C05492=1189.605,68.219,-48.419,-179.170,5.909,148.807
C05493=1189.600,68.469,-48.436,-179.167,5.909,148.806
C05494=1189.595,68.718,-48.452,-179.164,5.911,148.806
C05495=1189.590,68.967,-48.469,-179.162,5.911,148.805
C05496=1189.585,69.217,-48.486,-179.160,5.912,148.805
C05497=1189.581,69.466,-48.504,-179.157,5.913,148.804
C05498=1189.575,69.715,-48.520,-179.154,5.914,148.804
C05499=1189.570,69.965,-48.538,-179.152,5.915,148.803
C05500=1189.566,70.214,-48.554,-179.149,5.916,148.802
C05501=1189.561,70.464,-48.572,-179.146,5.917,148.802
C05502=1189.555,70.713,-48.588,-179.144,5.918,148.801
C05503=1189.551,70.962,-48.604,-179.142,5.919,148.801
C05504=1189.546,71.211,-48.622,-179.138,5.920,148.800
C05505=1189.542,71.461,-48.639,-179.136,5.921,148.800
C05506=1189.536,71.710,-48.656,-179.134,5.922,148.799
C05507=1189.531,71.960,-48.673,-179.130,5.923,148.798
C05508=1189.526,72.209,-48.690,-179.128,5.924,148.798
C05509=1189.521,72.458,-48.708,-179.126,5.924,148.797
C05510=1189.517,72.708,-48.725,-179.123,5.926,148.797
C05511=1189.511,72.957,-48.742,-179.120,5.927,148.796
C05512=1189.506,73.206,-48.758,-179.118,5.927,148.796
C05513=1189.501,73.456,-48.776,-179.115,5.928,148.795
C05514=1189.497,73.705,-48.793,-179.112,5.929,148.794
C05515=1189.492,73.955,-48.810,-179.110,5.930,148.794
C05516=1189.487,74.204,-48.827,-179.107,5.931,148.793
C05517=1189.482,74.453,-48.844,-179.105,5.933,148.793
C05518=1189.477,74.703,-48.862,-179.102,5.933,148.792
C05519=1189.472,74.952,-48.878,-179.100,5.934,148.792
C05520=1189.467,75.201,-48.896,-179.097,5.935,148.791
C05521=1189.463,75.451,-48.913,-179.094,5.936,148.791
C05522=1189.457,75.701,-48.930,-179.092,5.937,148.790
C05523=1189.453,75.950,-48.948,-179.089,5.938,148.789
C05524=1189.447,76.199,-48.965,-179.087,5.939,148.789
C05525=1189.442,76.448,-48.982,-179.084,5.940,148.788
C05526=1189.438,76.697,-48.999,-179.081,5.941,148.788
C05527=1189.433,76.947,-49.016,-179.079,5.942,148.787
C05528=1189.428,77.196,-49.034,-179.076,5.944,148.787
C05529=1189.423,77.446,-49.051,-179.073,5.944,148.786
C05530=1189.419,77.695,-49.069,-179.071,5.945,148.786
C05531=1189.413,77.945,-49.086,-179.068,5.946,148.785
C05532=1189.408,78.193,-49.103,-179.065,5.947,148.784
C05533=1189.403,78.443,-49.121,-179.063,5.948,148.784
C05534=1189.398,78.692,-49.138,-179.060,5.949,148.783
C05535=1189.394,78.941,-49.155,-179.058,5.950,148.783
C05536=1189.389,79.191,-49.173,-179.055,5.951,148.782
C05537=1189.384,79.440,-49.190,-179.053,5.952,148.782
C05538=1189.379,79.690,-49.208,-179.050,5.953,148.781
C05539=1189.374,79.939,-49.225,-179.048,5.954,148.781
C05540=1189.369,80.189,-49.242,-179.045,5.955,148.780
C05541=1189.364,80.457,-49.262,-179.042,5.956,148.780
C05542=1189.358,80.725,-49.280,-179.039,5.957,148.779
C05543=1189.354,80.994,-49.298,-179.037,5.958,148.778
C05544=1189.348,81.262,-49.318,-179.033,5.959,148.778
C05545=1189.344,81.511,-49.336,-179.031,5.960,148.777
C05546=1189.338,81.761,-49.353,-179.028,5.962,148.777
C05547=1189.333,82.010,-49.371,-179.026,5.963,148.776
C05548=1189.329,82.260,-49.388,-179.023,5.963,148.776
C05549=1189.324,82.509,-49.406,-179.020,5.964,148.775
C05550=1189.319,82.759,-49.423,-179.018,5.965,148.775
C05551=1189.314,83.008,-49.441,-179.015,5.967,148.774
C05552=1189.309,83.257,-49.459,-179.013,5.968,148.773
C05553=1189.304,83.506,-49.475,-179.010,5.968,148.773
C05554=1189.300,83.756,-49.493,-179.007,5.970,148.772
C05555=1189.295,84.005,-49.511,-179.005,5.970,148.772
C05556=1189.289,84.255,-49.529,-179.002,5.972,148.771
C05557=1189.285,84.504,-49.547,-178.999,5.973,148.771
C05558=1189.280,84.753,-49.565,-178.997,5.974,148.770
C05559=1189.275,85.002,-49.581,-178.994,5.975,148.770
C05560=1189.270,85.252,-49.599,-178.992,5.976,148.769
C05561=1189.265,85.501,-49.617,-178.989,5.977,148.769
C05562=1189.260,85.750,-49.635,-178.986,5.978,148.768
C05563=1189.255,86.000,-49.652,-178.984,5.979,148.767
C05564=1189.250,86.249,-49.670,-178.981,5.980,148.767
C05565=1189.245,86.498,-49.688,-178.979,5.981,148.766
C05566=1189.240,86.747,-49.706,-178.976,5.983,148.766
C05567=1189.236,86.997,-49.723,-178.973,5.983,148.765
C05568=1189.231,87.246,-49.741,-178.971,5.984,148.765
C05569=1189.226,87.495,-49.759,-178.968,5.986,148.764
C05570=1189.221,87.744,-49.777,-178.966,5.986,148.764
C05571=1189.216,87.993,-49.795,-178.962,5.988,148.763
C05572=1189.211,88.243,-49.812,-178.960,5.989,148.763
C05573=1189.206,88.492,-49.830,-178.958,5.989,148.762
C05574=1189.201,88.742,-49.848,-178.955,5.991,148.762
C05575=1189.196,88.991,-49.866,-178.952,5.992,148.761
C05576=1189.191,89.240,-49.884,-178.950,5.993,148.761
C05577=1189.187,89.490,-49.903,-178.947,5.994,148.760
C05578=1189.182,89.740,-49.920,-178.944,5.996,148.760
C05579=1189.177,89.989,-49.938,-178.942,5.996,148.759
C05580=1189.172,90.238,-49.956,-178.940,5.997,148.758
C05581=1189.167,90.487,-49.974,-178.936,5.998,148.758
C05582=1189.162,90.736,-49.992,-178.934,5.999,148.757
C05583=1189.157,90.985,-50.010,-178.931,6.001,148.757
C05584=1189.152,91.235,-50.028,-178.929,6.002,148.756
C05585=1189.148,91.484,-50.046,-178.926,6.003,148.756
C05586=1189.143,91.734,-50.064,-178.924,6.004,148.755
C05587=1189.138,91.983,-50.082,-178.921,6.004,148.755
C05588=1189.133,92.232,-50.100,-178.918,6.006,148.754
C05589=1189.128,92.481,-50.118,-178.916,6.007,148.754
C05590=1189.124,92.730,-50.136,-178.913,6.008,148.753
C05591=1189.119,92.980,-50.154,-178.910,6.009,148.753
C05592=1189.114,93.229,-50.172,-178.908,6.011,148.752
C05593=1189.109,93.479,-50.190,-178.905,6.011,148.751
C05594=1189.105,93.728,-50.208,-178.902,6.013,148.751
C05595=1189.100,93.977,-50.226,-178.900,6.014,148.750
C05596=1189.095,94.226,-50.244,-178.897,6.015,148.750
C05597=1189.089,94.476,-50.263,-178.895,6.016,148.750
C05598=1189.084,94.725,-50.281,-178.892,6.017,148.749
C05599=1189.080,94.975,-50.299,-178.889,6.019,148.748
C05600=1189.075,95.224,-50.317,-178.887,6.019,148.748
C05601=1189.070,95.473,-50.335,-178.884,6.021,148.747
C05602=1189.065,95.722,-50.353,-178.881,6.021,148.747
C05603=1189.060,95.971,-50.372,-178.879,6.023,148.746
C05604=1189.055,96.221,-50.391,-178.876,6.024,148.746
C05605=1189.051,96.470,-50.409,-178.873,6.025,148.745
C05606=1189.046,96.719,-50.427,-178.871,6.026,148.745
C05607=1189.041,96.968,-50.445,-178.869,6.027,148.744
C05608=1189.036,97.218,-50.463,-178.865,6.028,148.744
C05609=1189.031,97.467,-50.481,-178.863,6.029,148.743
C05610=1189.026,97.716,-50.500,-178.861,6.031,148.743
C05611=1189.021,97.966,-50.518,-178.858,6.032,148.742
C05612=1189.016,98.215,-50.536,-178.855,6.033,148.742
C05613=1189.012,98.465,-50.555,-178.853,6.034,148.741
C05614=1189.007,98.714,-50.572,-178.850,6.036,148.741
C05615=1189.002,98.963,-50.592,-178.847,6.036,148.740
C05616=1188.997,99.212,-50.610,-178.845,6.038,148.740
C05617=1188.993,99.462,-50.628,-178.842,6.038,148.739
C05618=1188.988,99.711,-50.646,-178.839,6.040,148.739
C05619=1188.982,99.960,-50.665,-178.837,6.041,148.738
C05620=1188.977,100.209,-50.683,-178.834,6.042,148.737
C05621=1188.973,100.459,-50.702,-178.832,6.043,148.737
C05622=1188.968,100.707,-50.720,-178.829,6.045,148.736
C05623=1188.963,100.957,-50.739,-178.827,6.046,148.736
C05624=1188.958,101.207,-50.757,-178.823,6.047,148.735
C05625=1188.954,101.455,-50.776,-178.821,6.048,148.735
C05626=1188.949,101.704,-50.794,-178.818,6.049,148.734
C05627=1188.944,101.955,-50.813,-178.816,6.050,148.734
C05628=1188.939,102.203,-50.832,-178.813,6.052,148.733
C05629=1188.934,102.452,-50.850,-178.811,6.053,148.733
C05630=1188.929,102.702,-50.868,-178.808,6.054,148.732
C05631=1188.925,102.951,-50.887,-178.805,6.055,148.732
C05632=1188.920,103.200,-50.905,-178.803,6.057,148.731
C05633=1188.914,103.449,-50.925,-178.800,6.057,148.731
C05634=1188.910,103.699,-50.943,-178.797,6.059,148.730
C05635=1188.905,103.948,-50.961,-178.795,6.060,148.730
C05636=1188.900,104.197,-50.980,-178.792,6.061,148.729
C05637=1188.896,104.447,-50.998,-178.790,6.062,148.729
C05638=1188.890,104.696,-51.018,-178.787,6.064,148.728
C05639=1188.885,104.945,-51.036,-178.784,6.064,148.728
C05640=1188.881,105.194,-51.055,-178.781,6.066,148.727
C05641=1188.876,105.444,-51.073,-178.779,6.067,148.727
C05642=1188.872,105.693,-51.092,-178.776,6.068,148.726
C05643=1188.866,105.942,-51.111,-178.774,6.069,148.726
C05644=1188.861,106.191,-51.130,-178.771,6.071,148.725
C05645=1188.856,106.460,-51.150,-178.768,6.072,148.725
C05646=1188.851,106.728,-51.170,-178.766,6.073,148.724
C05647=1188.846,106.996,-51.190,-178.763,6.074,148.724
C05648=1188.841,107.265,-51.210,-178.759,6.076,148.723
C05649=1188.836,107.514,-51.229,-178.757,6.077,148.723
C05650=1188.831,107.763,-51.248,-178.755,6.079,148.722
C05651=1188.826,108.013,-51.267,-178.752,6.079,148.722
C05652=1188.822,108.262,-51.286,-178.749,6.081,148.721
C05653=1188.816,108.512,-51.305,-178.747,6.081,148.720
C05654=1188.812,108.760,-51.323,-178.744,6.083,148.720
C05655=1188.807,109.010,-51.343,-178.741,6.085,148.720
C05656=1188.802,109.259,-51.361,-178.739,6.085,148.719
C05657=1188.797,109.508,-51.380,-178.736,6.087,148.719
C05658=1188.793,109.757,-51.399,-178.733,6.088,148.718
C05659=1188.787,110.007,-51.418,-178.731,6.090,148.718
C05660=1188.783,110.256,-51.437,-178.728,6.090,148.717
C05661=1188.778,110.505,-51.456,-178.725,6.092,148.717
C05662=1188.774,110.755,-51.474,-178.723,6.093,148.716
C05663=1188.768,111.004,-51.494,-178.720,6.094,148.716
C05664=1188.764,111.253,-51.513,-178.717,6.096,148.715
C05665=1188.759,111.502,-51.531,-178.715,6.097,148.715
C05666=1188.754,111.752,-51.551,-178.712,6.098,148.714
C05667=1188.749,112.000,-51.570,-178.710,6.099,148.714
C05668=1188.744,112.250,-51.589,-178.707,6.101,148.713
C05669=1188.740,112.499,-51.607,-178.704,6.101,148.713
C05670=1188.735,112.749,-51.627,-178.702,6.103,148.712
C05671=1188.729,112.998,-51.646,-178.699,6.104,148.712
C05672=1188.725,113.247,-51.665,-178.696,6.106,148.711
C05673=1188.720,113.496,-51.685,-178.694,6.107,148.711
C05674=1188.716,113.746,-51.703,-178.691,6.108,148.710
C05675=1188.710,113.994,-51.722,-178.688,6.110,148.710
C05676=1188.706,114.244,-51.742,-178.686,6.111,148.709
C05677=1188.701,114.493,-51.761,-178.683,6.112,148.709
C05678=1188.696,114.742,-51.780,-178.680,6.114,148.708
C05679=1188.691,114.991,-51.800,-178.678,6.114,148.708
C05680=1188.687,115.240,-51.819,-178.675,6.116,148.707
C05681=1188.681,115.490,-51.837,-178.673,6.117,148.707
C05682=1188.677,115.739,-51.857,-178.670,6.118,148.706
C05683=1188.672,115.988,-51.876,-178.668,6.119,148.706
C05684=1188.667,116.237,-51.895,-178.665,6.121,148.705
C05685=1188.662,116.486,-51.915,-178.662,6.122,148.705
C05686=1188.658,116.736,-51.934,-178.660,6.123,148.704
C05687=1188.653,116.985,-51.953,-178.657,6.125,148.704
C05688=1188.648,117.234,-51.973,-178.654,6.126,148.703
C05689=1188.643,117.484,-51.992,-178.652,6.127,148.703
C05690=1188.638,117.732,-52.011,-178.649,6.129,148.703
C05691=1188.634,117.982,-52.031,-178.646,6.130,148.702
C05692=1188.628,118.231,-52.050,-178.644,6.131,148.701
C05693=1188.624,118.480,-52.070,-178.641,6.132,148.701
C05694=1188.620,118.729,-52.089,-178.638,6.134,148.700
C05695=1188.614,118.978,-52.108,-178.636,6.136,148.700
C05696=1188.610,119.228,-52.128,-178.633,6.136,148.700
C05697=1188.604,119.477,-52.147,-178.630,6.138,148.699
C05698=1188.600,119.726,-52.166,-178.628,6.139,148.699
C05699=1188.595,119.976,-52.186,-178.625,6.141,148.698
C05700=1188.590,120.224,-52.205,-178.622,6.142,148.698
C05701=1188.585,120.474,-52.225,-178.620,6.143,148.697
C05702=1188.581,120.724,-52.244,-178.617,6.145,148.697
C05703=1188.575,120.972,-52.263,-178.614,6.146,148.696
C05704=1188.572,121.221,-52.283,-178.612,6.147,148.696
C05705=1188.566,121.470,-52.303,-178.609,6.149,148.695
C05706=1188.562,121.720,-52.322,-178.607,6.149,148.695
C05707=1188.557,121.969,-52.342,-178.604,6.151,148.694
C05708=1188.551,122.218,-52.361,-178.601,6.153,148.694
C05709=1188.547,122.468,-52.381,-178.599,6.153,148.693
C05710=1188.543,122.717,-52.400,-178.596,6.155,148.693
C05711=1188.538,122.965,-52.420,-178.593,6.157,148.692
C05712=1188.533,123.215,-52.440,-178.591,6.157,148.692
C05713=1188.528,123.464,-52.459,-178.588,6.159,148.691
C05714=1188.523,123.714,-52.479,-178.585,6.161,148.691
C05715=1188.518,123.962,-52.499,-178.583,6.162,148.690
C05716=1188.514,124.212,-52.518,-178.580,6.163,148.690
C05717=1188.509,124.461,-52.538,-178.578,6.164,148.690
C05718=1188.504,124.710,-52.557,-178.575,6.166,148.689
C05719=1188.499,124.959,-52.578,-178.572,6.167,148.689
C05720=1188.494,125.208,-52.597,-178.570,6.168,148.688
C05721=1188.490,125.457,-52.616,-178.567,6.170,148.688
C05722=1188.485,125.707,-52.636,-178.564,6.171,148.687
C05723=1188.481,125.956,-52.656,-178.562,6.172,148.687
C05724=1188.476,126.205,-52.676,-178.559,6.174,148.686
C05725=1188.470,126.454,-52.695,-178.556,6.176,148.686
C05726=1188.466,126.703,-52.715,-178.554,6.176,148.685
C05727=1188.461,126.953,-52.735,-178.551,6.178,148.685
C05728=1188.457,127.202,-52.755,-178.548,6.180,148.684
C05729=1188.452,127.450,-52.775,-178.546,6.181,148.684
C05730=1188.447,127.700,-52.794,-178.543,6.182,148.684
C05731=1188.442,127.949,-52.815,-178.540,6.184,148.683
C05732=1188.438,128.198,-52.834,-178.538,6.185,148.683
C05733=1188.432,128.447,-52.854,-178.535,6.186,148.682
C05734=1188.428,128.696,-52.874,-178.533,6.188,148.682
C05735=1188.423,128.946,-52.894,-178.530,6.189,148.681
C05736=1188.419,129.195,-52.914,-178.527,6.190,148.681
C05737=1188.414,129.444,-52.934,-178.525,6.192,148.680
C05738=1188.408,129.693,-52.954,-178.522,6.193,148.680
C05739=1188.403,129.942,-52.974,-178.519,6.195,148.679
C05740=1188.399,130.191,-52.994,-178.517,6.196,148.679
C05741=1188.394,130.441,-53.014,-178.515,6.197,148.679
C05742=1188.390,130.690,-53.035,-178.511,6.199,148.678
C05743=1188.384,130.939,-53.054,-178.509,6.200,148.678
C05744=1188.380,131.188,-53.074,-178.507,6.201,148.677
C05745=1188.375,131.437,-53.094,-178.504,6.203,148.677
C05746=1188.371,131.686,-53.114,-178.501,6.205,148.676
C05747=1188.366,131.936,-53.134,-178.498,6.206,148.676
C05748=1188.361,132.185,-53.155,-178.496,6.207,148.675
C05749=1188.356,132.454,-53.176,-178.493,6.209,148.675
C05750=1188.351,132.722,-53.198,-178.490,6.210,148.674
C05751=1188.346,132.991,-53.219,-178.487,6.212,148.674
C05752=1188.340,133.260,-53.241,-178.484,6.214,148.673
C05753=1188.336,133.509,-53.261,-178.481,6.215,148.673
C05754=1188.331,133.757,-53.281,-178.479,6.216,148.673
C05755=1188.326,134.006,-53.301,-178.476,6.218,148.672
C05756=1188.321,134.255,-53.321,-178.473,6.219,148.672
C05757=1188.316,134.505,-53.342,-178.471,6.220,148.671
C05758=1188.311,134.754,-53.362,-178.469,6.222,148.671
C05759=1188.307,135.003,-53.382,-178.465,6.224,148.670
C05760=1188.303,135.252,-53.403,-178.463,6.225,148.670
C05761=1188.298,135.502,-53.422,-178.461,6.226,148.669
C05762=1188.293,135.751,-53.443,-178.458,6.228,148.669
C05763=1188.288,135.999,-53.463,-178.455,6.229,148.668
C05764=1188.283,136.249,-53.483,-178.453,6.230,148.668
C05765=1188.278,136.498,-53.503,-178.450,6.232,148.668
C05766=1188.273,136.747,-53.524,-178.447,6.234,148.667
C05767=1188.269,136.996,-53.545,-178.444,6.235,148.667
C05768=1188.264,137.245,-53.564,-178.442,6.236,148.666
C05769=1188.259,137.495,-53.585,-178.439,6.238,148.666
C05770=1188.255,137.744,-53.606,-178.437,6.240,148.665
C05771=1188.250,137.993,-53.626,-178.433,6.241,148.665
C05772=1188.246,138.242,-53.647,-178.431,6.242,148.664
C05773=1188.240,138.491,-53.668,-178.429,6.244,148.664
C05774=1188.236,138.740,-53.687,-178.426,6.246,148.664
C05775=1188.231,138.989,-53.708,-178.423,6.246,148.663
C05776=1188.226,139.239,-53.729,-178.421,6.248,148.663
C05777=1188.222,139.488,-53.749,-178.418,6.250,148.662
C05778=1188.217,139.737,-53.769,-178.415,6.252,148.662
C05779=1188.212,139.986,-53.790,-178.413,6.252,148.661
C05780=1188.208,140.235,-53.811,-178.410,6.254,148.661
C05781=1188.202,140.484,-53.832,-178.407,6.256,148.660
C05782=1188.198,140.734,-53.851,-178.405,6.257,148.660
C05783=1188.193,140.983,-53.872,-178.402,6.258,148.660
C05784=1188.188,141.232,-53.893,-178.400,6.260,148.659
C05785=1188.184,141.481,-53.913,-178.397,6.262,148.659
C05786=1188.179,141.730,-53.933,-178.394,6.263,148.658
C05787=1188.174,141.979,-53.954,-178.392,6.264,148.658
C05788=1188.170,142.228,-53.975,-178.389,6.266,148.657
C05789=1188.164,142.477,-53.996,-178.386,6.268,148.657
C05790=1188.160,142.726,-54.016,-178.383,6.269,148.656
C05791=1188.155,142.975,-54.037,-178.381,6.271,148.656
C05792=1188.150,143.224,-54.057,-178.378,6.272,148.656
C05793=1188.146,143.473,-54.078,-178.376,6.274,148.655
C05794=1188.141,143.723,-54.099,-178.373,6.275,148.655
C05795=1188.136,143.971,-54.119,-178.370,6.277,148.654
C05796=1188.131,144.221,-54.140,-178.368,6.278,148.654
C05797=1188.127,144.469,-54.161,-178.365,6.280,148.654
C05798=1188.122,144.718,-54.182,-178.362,6.281,148.653
C05799=1188.117,144.967,-54.202,-178.360,6.283,148.653
C05800=1188.112,145.217,-54.223,-178.357,6.285,148.652
C05801=1188.108,145.465,-54.244,-178.354,6.285,148.652
C05802=1188.103,145.715,-54.265,-178.352,6.287,148.651
C05803=1188.099,145.964,-54.285,-178.349,6.289,148.651
C05804=1188.094,146.214,-54.306,-178.346,6.291,148.651
C05805=1188.089,146.463,-54.327,-178.344,6.292,148.650
C05806=1188.084,146.711,-54.349,-178.341,6.293,148.650
C05807=1188.079,146.960,-54.369,-178.338,6.295,148.649
C05808=1188.075,147.209,-54.390,-178.336,6.297,148.649
C05809=1188.070,147.459,-54.411,-178.333,6.298,148.648
C05810=1188.065,147.708,-54.431,-178.331,6.299,148.648
C05811=1188.060,147.956,-54.453,-178.328,6.301,148.647
C05812=1188.056,148.206,-54.474,-178.325,6.303,148.647
C05813=1188.051,148.455,-54.495,-178.322,6.304,148.647
C05814=1188.046,148.704,-54.516,-178.320,6.306,148.646
C05815=1188.042,148.953,-54.537,-178.318,6.307,148.646
C05816=1188.037,149.202,-54.558,-178.315,6.309,148.646
C05817=1188.032,149.451,-54.578,-178.312,6.311,148.645
C05818=1188.027,149.700,-54.600,-178.309,6.312,148.645
C05819=1188.023,149.950,-54.621,-178.306,6.314,148.644
C05820=1188.018,150.199,-54.641,-178.304,6.316,148.644
C05821=1188.013,150.448,-54.662,-178.302,6.316,148.643
C05822=1188.008,150.696,-54.684,-178.299,6.318,148.643
C05823=1188.004,150.945,-54.704,-178.296,6.320,148.643
C05824=1187.999,151.194,-54.726,-178.293,6.321,148.642
C05825=1187.994,151.444,-54.747,-178.290,6.323,148.642
C05826=1187.990,151.693,-54.768,-178.288,6.324,148.641
C05827=1187.985,151.942,-54.789,-178.285,6.326,148.641
C05828=1187.980,152.191,-54.810,-178.283,6.328,148.641
C05829=1187.975,152.440,-54.831,-178.280,6.329,148.640
C05830=1187.971,152.689,-54.853,-178.277,6.331,148.640
C05831=1187.966,152.938,-54.874,-178.274,6.333,148.639
C05832=1187.961,153.187,-54.895,-178.272,6.334,148.639
C05833=1187.956,153.436,-54.916,-178.269,6.335,148.638
C05834=1187.952,153.685,-54.938,-178.267,6.337,148.638
C05835=1187.947,153.935,-54.959,-178.264,6.339,148.638
C05836=1187.942,154.183,-54.981,-178.261,6.341,148.637
C05837=1187.937,154.432,-55.002,-178.259,6.342,148.637
C05838=1187.933,154.681,-55.023,-178.257,6.343,148.636
C05839=1187.929,154.931,-55.044,-178.253,6.345,148.636
C05840=1187.924,155.179,-55.066,-178.251,6.347,148.636
C05841=1187.919,155.429,-55.087,-178.248,6.348,148.635
C05842=1187.914,155.677,-55.108,-178.245,6.350,148.635
C05843=1187.910,155.927,-55.129,-178.243,6.352,148.634
C05844=1187.905,156.176,-55.151,-178.240,6.354,148.634
C05845=1187.900,156.424,-55.172,-178.238,6.355,148.634
C05846=1187.896,156.674,-55.194,-178.235,6.356,148.633
C05847=1187.891,156.923,-55.215,-178.233,6.358,148.633
C05848=1187.886,157.172,-55.236,-178.229,6.360,148.632
C05849=1187.881,157.420,-55.257,-178.227,6.361,148.632
C05850=1187.877,157.670,-55.279,-178.224,6.363,148.632
C05851=1187.872,157.919,-55.300,-178.221,6.365,148.631
C05852=1187.867,158.168,-55.322,-178.219,6.367,148.631
C05853=1187.862,158.437,-55.345,-178.216,6.369,148.630
C05854=1187.857,158.706,-55.368,-178.213,6.370,148.630
C05855=1187.852,158.975,-55.392,-178.210,6.372,148.629
C05856=1187.847,159.244,-55.415,-178.207,6.374,148.629
C05857=1187.842,159.492,-55.437,-178.205,6.375,148.629
C05858=1187.838,159.742,-55.459,-178.202,6.377,148.628
C05859=1187.833,159.991,-55.480,-178.199,6.379,148.628
C05860=1187.828,160.240,-55.501,-178.197,6.380,148.628
C05861=1187.823,160.489,-55.524,-178.195,6.382,148.627
C05862=1187.819,160.738,-55.545,-178.191,6.383,148.627
C05863=1187.814,160.988,-55.567,-178.189,6.385,148.626
C05864=1187.809,161.236,-55.588,-178.186,6.387,148.626
C05865=1187.804,161.485,-55.610,-178.183,6.388,148.625
C05866=1187.800,161.734,-55.632,-178.181,6.390,148.625
C05867=1187.795,161.983,-55.654,-178.178,6.392,148.625
C05868=1187.790,162.232,-55.675,-178.175,6.394,148.624
C05869=1187.786,162.482,-55.697,-178.173,6.395,148.624
C05870=1187.781,162.730,-55.718,-178.171,6.396,148.624
C05871=1187.777,162.980,-55.740,-178.168,6.398,148.623
C05872=1187.772,163.228,-55.762,-178.165,6.400,148.623
C05873=1187.767,163.477,-55.784,-178.163,6.402,148.622
C05874=1187.763,163.726,-55.806,-178.160,6.404,148.622
C05875=1187.758,163.975,-55.827,-178.157,6.405,148.622
C05876=1187.753,164.225,-55.849,-178.154,6.407,148.621
C05877=1187.748,164.473,-55.870,-178.151,6.408,148.621
C05878=1187.744,164.723,-55.893,-178.149,6.410,148.620
C05879=1187.739,164.971,-55.914,-178.146,6.412,148.620
C05880=1187.734,165.220,-55.936,-178.144,6.413,148.620
C05881=1187.730,165.469,-55.958,-178.141,6.415,148.619
C05882=1187.725,165.718,-55.980,-178.139,6.417,148.619
C05883=1187.721,165.967,-56.002,-178.136,6.418,148.619
C05884=1187.716,166.216,-56.023,-178.133,6.420,148.618
C05885=1187.712,166.465,-56.045,-178.131,6.422,148.618
C05886=1187.706,166.714,-56.068,-178.128,6.424,148.617
C05887=1187.702,166.964,-56.090,-178.125,6.425,148.617
C05888=1187.697,167.212,-56.111,-178.123,6.427,148.617
C05889=1187.693,167.462,-56.133,-178.120,6.429,148.616
C05890=1187.688,167.710,-56.156,-178.117,6.431,148.616
C05891=1187.684,167.959,-56.178,-178.114,6.433,148.616
C05892=1187.678,168.208,-56.200,-178.112,6.434,148.615
C05893=1187.674,168.457,-56.222,-178.109,6.436,148.615
C05894=1187.669,168.706,-56.244,-178.107,6.437,148.615
C05895=1187.665,168.955,-56.266,-178.104,6.439,148.614
C05896=1187.660,169.204,-56.288,-178.102,6.441,148.614
C05897=1187.655,169.454,-56.310,-178.099,6.442,148.613
C05898=1187.650,169.702,-56.332,-178.096,6.444,148.613
C05899=1187.646,169.951,-56.355,-178.094,6.446,148.613
C05900=1187.641,170.200,-56.376,-178.090,6.447,148.612
C05901=1187.637,170.449,-56.398,-178.088,6.449,148.612
C05902=1187.631,170.698,-56.421,-178.085,6.451,148.611
C05903=1187.627,170.947,-56.443,-178.082,6.453,148.611
C05904=1187.623,171.195,-56.465,-178.080,6.455,148.611
C05905=1187.618,171.445,-56.488,-178.077,6.456,148.610
C05906=1187.613,171.694,-56.510,-178.074,6.458,148.610
C05907=1187.608,171.943,-56.532,-178.072,6.460,148.610
C05908=1187.604,172.192,-56.554,-178.069,6.462,148.609
C05909=1187.599,172.440,-56.577,-178.066,6.464,148.609
C05910=1187.595,172.690,-56.599,-178.064,6.465,148.608
C05911=1187.590,172.938,-56.621,-178.061,6.467,148.608
C05912=1187.585,173.187,-56.644,-178.058,6.469,148.608
C05913=1187.581,173.437,-56.666,-178.056,6.471,148.607
C05914=1187.576,173.685,-56.688,-178.053,6.472,148.607
C05915=1187.571,173.935,-56.711,-178.050,6.474,148.607
C05916=1187.566,174.183,-56.732,-178.048,6.476,148.606
C05917=1187.562,174.432,-56.755,-178.045,6.478,148.606
C05918=1187.557,174.682,-56.778,-178.042,6.480,148.606
C05919=1187.552,174.930,-56.800,-178.040,6.481,148.605
C05920=1187.549,175.179,-56.822,-178.037,6.483,148.605
C05921=1187.544,175.429,-56.845,-178.034,6.485,148.604
C05922=1187.539,175.677,-56.867,-178.032,6.487,148.604
C05923=1187.534,175.926,-56.890,-178.029,6.489,148.604
C05924=1187.529,176.175,-56.912,-178.027,6.491,148.604
C05925=1187.524,176.424,-56.935,-178.024,6.492,148.603
C05926=1187.520,176.673,-56.957,-178.021,6.494,148.603
C05927=1187.516,176.921,-56.980,-178.019,6.496,148.603
C05928=1187.511,177.171,-57.002,-178.016,6.498,148.602
C05929=1187.507,177.420,-57.025,-178.013,6.500,148.602
C05930=1187.501,177.669,-57.047,-178.011,6.501,148.601
C05931=1187.497,177.917,-57.070,-178.008,6.503,148.601
C05932=1187.492,178.167,-57.093,-178.005,6.505,148.601
C05933=1187.487,178.415,-57.115,-178.003,6.507,148.600
C05934=1187.483,178.664,-57.138,-178.000,6.508,148.600
C05935=1187.478,178.913,-57.160,-177.997,6.510,148.600
C05936=1187.474,179.162,-57.184,-177.995,6.512,148.599
C05937=1187.469,179.411,-57.205,-177.992,6.514,148.599
C05938=1187.464,179.660,-57.229,-177.989,6.516,148.599
C05939=1187.460,179.909,-57.251,-177.987,6.517,148.598
C05940=1187.455,180.158,-57.274,-177.984,6.519,148.598
C05941=1187.451,180.406,-57.297,-177.981,6.521,148.597
C05942=1187.446,180.656,-57.319,-177.979,6.523,148.597
C05943=1187.442,180.905,-57.342,-177.976,6.525,148.597
C05944=1187.436,181.153,-57.365,-177.973,6.526,148.596
C05945=1187.432,181.402,-57.387,-177.971,6.528,148.596
C05946=1187.427,181.652,-57.410,-177.968,6.530,148.596
C05947=1187.423,181.900,-57.433,-177.966,6.532,148.596
C05948=1187.418,182.149,-57.456,-177.963,6.534,148.595
C05949=1187.413,182.398,-57.479,-177.960,6.536,148.595
C05950=1187.409,182.647,-57.502,-177.958,6.537,148.594
C05951=1187.404,182.896,-57.525,-177.955,6.539,148.594
C05952=1187.400,183.145,-57.547,-177.952,6.541,148.594
C05953=1187.395,183.394,-57.570,-177.950,6.543,148.593
C05954=1187.390,183.643,-57.593,-177.947,6.545,148.593
C05955=1187.386,183.891,-57.616,-177.944,6.546,148.593
C05956=1187.382,184.140,-57.639,-177.942,6.548,148.592
C05957=1187.376,184.410,-57.664,-177.939,6.550,148.592
C05958=1187.372,184.680,-57.689,-177.936,6.553,148.592
C05959=1187.366,184.949,-57.714,-177.933,6.554,148.591
C05960=1187.362,185.219,-57.738,-177.931,6.556,148.591
C05961=1187.357,185.468,-57.762,-177.928,6.558,148.591
C05962=1187.352,185.716,-57.785,-177.925,6.561,148.590
C05963=1187.347,185.965,-57.808,-177.922,6.562,148.590
C05964=1187.343,186.214,-57.831,-177.919,6.564,148.590
C05965=1187.338,186.464,-57.854,-177.917,6.566,148.589
C05966=1187.333,186.713,-57.877,-177.914,6.568,148.589
C05967=1187.329,186.961,-57.900,-177.912,6.570,148.589
C05968=1187.324,187.210,-57.923,-177.909,6.572,148.588
C05969=1187.319,187.459,-57.946,-177.906,6.573,148.588
C05970=1187.315,187.708,-57.969,-177.904,6.575,148.588
C05971=1187.311,187.956,-57.992,-177.901,6.577,148.587
C05972=1187.306,188.206,-58.015,-177.898,6.579,148.587
C05973=1187.301,188.455,-58.039,-177.896,6.581,148.587
C05974=1187.297,188.704,-58.062,-177.893,6.582,148.586
C05975=1187.292,188.953,-58.086,-177.890,6.584,148.586
C05976=1187.287,189.201,-58.108,-177.887,6.587,148.586
C05977=1187.283,189.450,-58.131,-177.885,6.589,148.585
C05978=1187.278,189.699,-58.155,-177.882,6.591,148.585
C05979=1187.273,189.948,-58.178,-177.880,6.593,148.585
C05980=1187.269,190.197,-58.201,-177.877,6.594,148.584
C05981=1187.264,190.446,-58.225,-177.874,6.596,148.584
C05982=1187.260,190.694,-58.248,-177.872,6.598,148.584
C05983=1187.256,190.943,-58.272,-177.869,6.600,148.583
C05984=1187.251,191.192,-58.295,-177.866,6.602,148.583
C05985=1187.246,191.441,-58.318,-177.864,6.604,148.583
C05986=1187.241,191.690,-58.342,-177.862,6.605,148.582
C05987=1187.237,191.939,-58.365,-177.858,6.608,148.582
C05988=1187.231,192.187,-58.388,-177.856,6.610,148.582
C05989=1187.227,192.436,-58.411,-177.853,6.612,148.581
C05990=1187.223,192.685,-58.435,-177.850,6.613,148.581
C05991=1187.218,192.934,-58.458,-177.848,6.615,148.581
C05992=1187.214,193.183,-58.482,-177.845,6.617,148.581
C05993=1187.209,193.432,-58.505,-177.843,6.619,148.580
C05994=1187.205,193.680,-58.529,-177.840,6.621,148.580
C05995=1187.200,193.929,-58.552,-177.837,6.623,148.580
C05996=1187.195,194.178,-58.576,-177.834,6.625,148.579
C05997=1187.191,194.427,-58.599,-177.832,6.627,148.579
C05998=1187.186,194.676,-58.623,-177.829,6.629,148.579
C05999=1187.181,194.925,-58.647,-177.827,6.631,148.578
C06000=1187.177,195.174,-58.670,-177.824,6.633,148.578
C06001=1187.172,195.423,-58.693,-177.821,6.635,148.578
C06002=1187.168,195.671,-58.717,-177.819,6.637,148.577
C06003=1187.163,195.920,-58.741,-177.816,6.638,148.577
C06004=1187.158,196.169,-58.764,-177.813,6.640,148.577
C06005=1187.154,196.418,-58.788,-177.811,6.643,148.577
C06006=1187.149,196.667,-58.811,-177.808,6.645,148.576
C06007=1187.145,196.915,-58.836,-177.805,6.647,148.576
C06008=1187.140,197.164,-58.859,-177.803,6.648,148.576
C06009=1187.135,197.413,-58.882,-177.800,6.650,148.575
C06010=1187.132,197.662,-58.907,-177.797,6.652,148.575
C06011=1187.127,197.911,-58.930,-177.795,6.654,148.575
C06012=1187.122,198.160,-58.954,-177.792,6.657,148.574
C06013=1187.118,198.409,-58.977,-177.789,6.659,148.574
C06014=1187.113,198.657,-59.002,-177.787,6.660,148.574
C06015=1187.108,198.906,-59.026,-177.784,6.662,148.573
C06016=1187.104,199.155,-59.050,-177.782,6.664,148.573
C06017=1187.099,199.404,-59.073,-177.779,6.666,148.573
C06018=1187.094,199.652,-59.097,-177.776,6.668,148.573
C06019=1187.090,199.901,-59.120,-177.773,6.671,148.572
C06020=1187.085,200.150,-59.144,-177.771,6.672,148.572
C06021=1187.081,200.399,-59.168,-177.768,6.674,148.572
C06022=1187.076,200.648,-59.193,-177.766,6.676,148.571
C06023=1187.071,200.897,-59.216,-177.763,6.678,148.571
C06024=1187.067,201.146,-59.240,-177.760,6.680,148.571
C06025=1187.062,201.395,-59.264,-177.757,6.683,148.570
C06026=1187.058,201.643,-59.288,-177.754,6.684,148.570
C06027=1187.054,201.891,-59.312,-177.752,6.687,148.570
C06028=1187.048,202.141,-59.336,-177.750,6.688,148.570
C06029=1187.044,202.389,-59.360,-177.747,6.690,148.569
C06030=1187.040,202.639,-59.384,-177.744,6.692,148.569
C06031=1187.035,202.887,-59.408,-177.742,6.695,148.569
C06032=1187.031,203.136,-59.432,-177.739,6.697,148.568
C06033=1187.026,203.384,-59.456,-177.736,6.698,148.568
C06034=1187.021,203.634,-59.480,-177.734,6.700,148.568
C06035=1187.017,203.882,-59.504,-177.731,6.702,148.567
C06036=1187.013,204.131,-59.528,-177.728,6.705,148.567
C06037=1187.007,204.380,-59.552,-177.726,6.707,148.567
C06038=1187.003,204.629,-59.576,-177.723,6.709,148.567
C06039=1186.999,204.877,-59.600,-177.720,6.710,148.566
C06040=1186.994,205.126,-59.624,-177.718,6.713,148.566
C06041=1186.989,205.376,-59.649,-177.715,6.715,148.566
C06042=1186.985,205.624,-59.673,-177.712,6.717,148.566
C06043=1186.981,205.873,-59.697,-177.709,6.719,148.565
C06044=1186.975,206.121,-59.722,-177.707,6.721,148.565
C06045=1186.971,206.370,-59.746,-177.705,6.723,148.565
C06046=1186.967,206.619,-59.769,-177.701,6.725,148.564
C06047=1186.962,206.868,-59.794,-177.699,6.727,148.564
C06048=1186.957,207.117,-59.818,-177.696,6.729,148.564
C06049=1186.953,207.365,-59.842,-177.694,6.731,148.564
C06050=1186.948,207.614,-59.867,-177.691,6.733,148.563
C06051=1186.944,207.863,-59.891,-177.688,6.736,148.563
C06052=1186.939,208.111,-59.916,-177.685,6.737,148.563
C06053=1186.934,208.361,-59.939,-177.683,6.740,148.562
C06054=1186.930,208.610,-59.964,-177.681,6.741,148.562
C06055=1186.925,208.858,-59.988,-177.678,6.743,148.562
C06056=1186.921,209.107,-60.012,-177.675,6.746,148.561
C06057=1186.916,209.355,-60.037,-177.672,6.748,148.561
C06058=1186.912,209.605,-60.062,-177.670,6.750,148.561
C06059=1186.907,209.853,-60.086,-177.667,6.752,148.561
C06060=1186.902,210.102,-60.110,-177.664,6.754,148.560
C06061=1186.898,210.373,-60.137,-177.662,6.756,148.560
C06062=1186.893,210.643,-60.164,-177.659,6.759,148.560
C06063=1186.888,210.913,-60.191,-177.656,6.761,148.560
C06064=1186.883,211.183,-60.216,-177.653,6.763,148.559
C06065=1186.878,211.433,-60.241,-177.650,6.765,148.559
C06066=1186.874,211.681,-60.266,-177.648,6.767,148.559
C06067=1186.869,211.929,-60.291,-177.645,6.769,148.558
C06068=1186.865,212.178,-60.315,-177.642,6.772,148.558
C06069=1186.860,212.427,-60.340,-177.639,6.774,148.558
C06070=1186.855,212.676,-60.365,-177.637,6.776,148.558
C06071=1186.851,212.925,-60.389,-177.634,6.778,148.557
C06072=1186.846,213.174,-60.414,-177.631,6.780,148.557
C06073=1186.842,213.422,-60.438,-177.629,6.782,148.557
C06074=1186.837,213.672,-60.463,-177.626,6.784,148.557
C06075=1186.833,213.919,-60.488,-177.624,6.786,148.556
C06076=1186.829,214.169,-60.513,-177.621,6.789,148.556
C06077=1186.824,214.417,-60.537,-177.618,6.791,148.556
C06078=1186.819,214.666,-60.561,-177.616,6.792,148.556
C06079=1186.815,214.915,-60.586,-177.613,6.794,148.555
C06080=1186.810,215.163,-60.611,-177.610,6.797,148.555
C06081=1186.805,215.412,-60.636,-177.608,6.799,148.555
C06082=1186.802,215.661,-60.660,-177.605,6.801,148.554
C06083=1186.796,215.910,-60.685,-177.603,6.803,148.554
C06084=1186.792,216.159,-60.711,-177.600,6.806,148.554
C06085=1186.788,216.407,-60.735,-177.597,6.807,148.554
C06086=1186.783,216.656,-60.760,-177.594,6.809,148.553
C06087=1186.778,216.904,-60.785,-177.592,6.811,148.553
C06088=1186.774,217.153,-60.809,-177.589,6.814,148.553
C06089=1186.770,217.402,-60.834,-177.586,6.816,148.553
C06090=1186.765,217.650,-60.860,-177.584,6.818,148.552
C06091=1186.761,217.900,-60.884,-177.581,6.821,148.552
C06092=1186.756,218.148,-60.909,-177.578,6.822,148.552
C06093=1186.752,218.397,-60.935,-177.576,6.825,148.552
C06094=1186.747,218.645,-60.959,-177.573,6.826,148.551
C06095=1186.743,218.895,-60.984,-177.570,6.829,148.551
C06096=1186.738,219.143,-61.009,-177.568,6.831,148.551
C06097=1186.733,219.392,-61.034,-177.565,6.833,148.551
C06098=1186.729,219.640,-61.059,-177.563,6.835,148.550
C06099=1186.724,219.889,-61.084,-177.560,6.838,148.550
C06100=1186.720,220.138,-61.109,-177.557,6.840,148.550
C06101=1186.715,220.386,-61.133,-177.555,6.841,148.550
C06102=1186.711,220.635,-61.159,-177.552,6.844,148.549
C06103=1186.706,220.884,-61.184,-177.549,6.846,148.549
C06104=1186.702,221.132,-61.209,-177.547,6.848,148.549
C06105=1186.697,221.382,-61.235,-177.544,6.851,148.549
C06106=1186.693,221.630,-61.259,-177.541,6.853,148.548
C06107=1186.689,221.879,-61.284,-177.539,6.855,148.548
C06108=1186.684,222.127,-61.310,-177.536,6.857,148.548
C06109=1186.679,222.377,-61.335,-177.533,6.859,148.548
C06110=1186.675,222.625,-61.360,-177.531,6.862,148.548
C06111=1186.670,222.874,-61.386,-177.528,6.863,148.547
C06112=1186.666,223.122,-61.410,-177.525,6.866,148.547
C06113=1186.662,223.371,-61.436,-177.523,6.868,148.547
C06114=1186.657,223.620,-61.460,-177.520,6.870,148.546
C06115=1186.652,223.868,-61.486,-177.518,6.873,148.546
C06116=1186.647,224.116,-61.512,-177.515,6.875,148.546
C06117=1186.643,224.366,-61.537,-177.512,6.877,148.546
C06118=1186.639,224.615,-61.562,-177.509,6.880,148.546
C06119=1186.634,224.863,-61.588,-177.507,6.881,148.545
C06120=1186.629,225.112,-61.613,-177.505,6.883,148.545
C06121=1186.625,225.360,-61.638,-177.501,6.886,148.545
C06122=1186.621,225.609,-61.663,-177.499,6.888,148.545
C06123=1186.617,225.858,-61.689,-177.497,6.890,148.544
C06124=1186.612,226.106,-61.714,-177.494,6.892,148.544
C06125=1186.607,226.355,-61.739,-177.491,6.895,148.544
C06126=1186.603,226.603,-61.765,-177.489,6.897,148.544
C06127=1186.598,226.852,-61.791,-177.486,6.899,148.543
C06128=1186.594,227.101,-61.816,-177.483,6.901,148.543
C06129=1186.589,227.350,-61.841,-177.481,6.903,148.543
C06130=1186.585,227.598,-61.867,-177.478,6.905,148.543
C06131=1186.580,227.846,-61.892,-177.475,6.908,148.543
C06132=1186.576,228.095,-61.918,-177.472,6.910,148.542
C06133=1186.572,228.344,-61.944,-177.470,6.913,148.542
C06134=1186.566,228.593,-61.968,-177.467,6.915,148.542
C06135=1186.562,228.842,-61.994,-177.465,6.917,148.542
C06136=1186.558,229.090,-62.020,-177.462,6.919,148.541
C06137=1186.553,229.338,-62.045,-177.460,6.922,148.541
C06138=1186.549,229.587,-62.071,-177.457,6.923,148.541
C06139=1186.545,229.836,-62.097,-177.454,6.926,148.541
C06140=1186.540,230.084,-62.122,-177.452,6.928,148.541
C06141=1186.536,230.333,-62.148,-177.449,6.930,148.540
C06142=1186.531,230.582,-62.174,-177.446,6.933,148.540
C06143=1186.526,230.831,-62.200,-177.443,6.935,148.540
C06144=1186.522,231.079,-62.225,-177.441,6.937,148.540
C06145=1186.517,231.328,-62.251,-177.438,6.940,148.540
C06146=1186.513,231.577,-62.277,-177.436,6.942,148.539
C06147=1186.508,231.825,-62.302,-177.433,6.944,148.539
C06148=1186.504,232.074,-62.328,-177.431,6.947,148.539
C06149=1186.500,232.322,-62.354,-177.428,6.948,148.539
C06150=1186.495,232.571,-62.380,-177.425,6.951,148.539
C06151=1186.490,232.820,-62.405,-177.422,6.953,148.538
C06152=1186.486,233.068,-62.431,-177.420,6.955,148.538
C06153=1186.482,233.317,-62.457,-177.417,6.958,148.538
C06154=1186.477,233.566,-62.483,-177.414,6.960,148.538
C06155=1186.473,233.814,-62.508,-177.412,6.962,148.537
C06156=1186.468,234.063,-62.534,-177.409,6.965,148.537
C06157=1186.464,234.311,-62.561,-177.407,6.967,148.537
C06158=1186.460,234.560,-62.587,-177.404,6.969,148.537
C06159=1186.455,234.808,-62.612,-177.402,6.972,148.537
C06160=1186.450,235.057,-62.638,-177.399,6.973,148.536
C06161=1186.446,235.306,-62.664,-177.396,6.976,148.536
C06162=1186.441,235.555,-62.690,-177.394,6.978,148.536
C06163=1186.437,235.803,-62.716,-177.391,6.981,148.536
C06164=1186.433,236.051,-62.742,-177.388,6.983,148.536
C06165=1186.427,236.324,-62.770,-177.385,6.986,148.536
C06166=1186.423,236.595,-62.799,-177.383,6.988,148.535
C06167=1186.418,236.867,-62.827,-177.380,6.990,148.535
C06168=1186.413,237.137,-62.856,-177.377,6.993,148.535
C06169=1186.408,237.386,-62.882,-177.374,6.995,148.535
C06170=1186.404,237.635,-62.908,-177.371,6.998,148.534
C06171=1186.400,237.883,-62.934,-177.369,7.000,148.534
C06172=1186.395,238.133,-62.960,-177.367,7.002,148.534
C06173=1186.391,238.381,-62.986,-177.363,7.005,148.534
C06174=1186.386,238.629,-63.012,-177.361,7.007,148.534
C06175=1186.381,238.878,-63.039,-177.358,7.010,148.533
C06176=1186.377,239.127,-63.064,-177.356,7.012,148.533
C06177=1186.372,239.375,-63.091,-177.354,7.014,148.533
C06178=1186.368,239.624,-63.117,-177.350,7.017,148.533
C06179=1186.364,239.872,-63.144,-177.348,7.019,148.533
C06180=1186.359,240.121,-63.170,-177.345,7.021,148.532
C06181=1186.354,240.369,-63.195,-177.343,7.024,148.532
C06182=1186.351,240.618,-63.222,-177.340,7.026,148.532
C06183=1186.346,240.867,-63.248,-177.338,7.028,148.532
C06184=1186.342,241.115,-63.275,-177.335,7.030,148.532
C06185=1186.337,241.364,-63.301,-177.332,7.033,148.532
C06186=1186.333,241.612,-63.328,-177.330,7.035,148.531
C06187=1186.328,241.861,-63.354,-177.327,7.038,148.531
C06188=1186.324,242.110,-63.380,-177.325,7.040,148.531
C06189=1186.319,242.359,-63.407,-177.321,7.043,148.531
C06190=1186.315,242.607,-63.433,-177.319,7.045,148.531
C06191=1186.311,242.856,-63.459,-177.317,7.047,148.530
C06192=1186.306,243.103,-63.486,-177.314,7.050,148.530
C06193=1186.302,243.352,-63.512,-177.311,7.052,148.530
C06194=1186.297,243.601,-63.538,-177.308,7.054,148.530
C06195=1186.293,243.849,-63.565,-177.306,7.057,148.530
C06196=1186.288,244.098,-63.591,-177.303,7.059,148.530
C06197=1186.283,244.347,-63.618,-177.301,7.061,148.530
C06198=1186.279,244.595,-63.645,-177.298,7.064,148.529
C06199=1186.274,244.844,-63.671,-177.296,7.066,148.529
C06200=1186.270,245.092,-63.698,-177.293,7.069,148.529
C06201=1186.266,245.340,-63.725,-177.290,7.071,148.529
C06202=1186.261,245.589,-63.750,-177.288,7.073,148.529
C06203=1186.257,245.838,-63.777,-177.285,7.076,148.528
C06204=1186.253,246.086,-63.804,-177.283,7.078,148.528
C06205=1186.248,246.335,-63.830,-177.280,7.081,148.528
C06206=1186.243,246.584,-63.857,-177.277,7.083,148.528
C06207=1186.239,246.832,-63.884,-177.275,7.086,148.528
C06208=1186.235,247.080,-63.911,-177.272,7.088,148.528
C06209=1186.230,247.329,-63.937,-177.269,7.091,148.527
C06210=1186.226,247.578,-63.964,-177.267,7.093,148.527
C06211=1186.221,247.826,-63.991,-177.264,7.095,148.527
C06212=1186.217,248.074,-64.017,-177.262,7.098,148.527
C06213=1186.213,248.323,-64.044,-177.259,7.101,148.527
C06214=1186.208,248.572,-64.071,-177.256,7.102,148.527
C06215=1186.204,248.820,-64.097,-177.254,7.105,148.527
C06216=1186.199,249.069,-64.124,-177.251,7.107,148.526
C06217=1186.194,249.317,-64.151,-177.248,7.110,148.526
C06218=1186.191,249.566,-64.178,-177.246,7.112,148.526
C06219=1186.186,249.814,-64.205,-177.243,7.115,148.526
C06220=1186.182,250.063,-64.232,-177.241,7.117,148.526
C06221=1186.177,250.311,-64.259,-177.238,7.120,148.526
C06222=1186.173,250.560,-64.286,-177.235,7.122,148.525
C06223=1186.168,250.809,-64.312,-177.233,7.125,148.525
C06224=1186.164,251.057,-64.339,-177.230,7.127,148.525
C06225=1186.160,251.305,-64.366,-177.227,7.130,148.525
C06226=1186.155,251.554,-64.393,-177.225,7.132,148.525
C06227=1186.150,251.802,-64.420,-177.222,7.135,148.525
C06228=1186.146,252.051,-64.447,-177.220,7.137,148.524
C06229=1186.142,252.300,-64.474,-177.217,7.140,148.524
C06230=1186.138,252.548,-64.501,-177.215,7.142,148.524
C06231=1186.133,252.797,-64.528,-177.212,7.145,148.524
C06232=1186.128,253.045,-64.555,-177.209,7.147,148.524
C06233=1186.124,253.293,-64.582,-177.207,7.150,148.524
C06234=1186.119,253.542,-64.610,-177.204,7.151,148.524
C06235=1186.115,253.790,-64.636,-177.201,7.154,148.524
C06236=1186.111,254.039,-64.663,-177.199,7.157,148.523
C06237=1186.107,254.287,-64.691,-177.196,7.159,148.523
C06238=1186.102,254.536,-64.718,-177.194,7.161,148.523
C06239=1186.097,254.784,-64.745,-177.191,7.164,148.523
C06240=1186.093,255.033,-64.772,-177.188,7.166,148.523
C06241=1186.088,255.281,-64.799,-177.186,7.169,148.523
C06242=1186.085,255.530,-64.826,-177.183,7.171,148.523
C06243=1186.080,255.778,-64.853,-177.181,7.174,148.522
C06244=1186.076,256.027,-64.880,-177.178,7.176,148.522
C06245=1186.071,256.275,-64.907,-177.175,7.179,148.522
C06246=1186.067,256.523,-64.935,-177.173,7.181,148.522
C06247=1186.063,256.772,-64.963,-177.170,7.184,148.522
C06248=1186.058,257.021,-64.990,-177.167,7.187,148.522
C06249=1186.053,257.269,-65.017,-177.165,7.189,148.522
C06250=1186.049,257.517,-65.045,-177.162,7.192,148.522
C06251=1186.044,257.766,-65.072,-177.160,7.194,148.521
C06252=1186.040,258.015,-65.099,-177.157,7.197,148.521
C06253=1186.036,258.263,-65.126,-177.155,7.199,148.521
C06254=1186.031,258.511,-65.154,-177.152,7.202,148.521
C06255=1186.027,258.760,-65.181,-177.150,7.204,148.521
C06256=1186.023,259.009,-65.208,-177.147,7.207,148.521
C06257=1186.018,259.257,-65.236,-177.144,7.210,148.521
C06258=1186.014,259.505,-65.263,-177.141,7.212,148.520
C06259=1186.009,259.753,-65.291,-177.139,7.215,148.520
C06260=1186.005,260.002,-65.318,-177.137,7.217,148.520
C06261=1186.001,260.251,-65.346,-177.134,7.220,148.520
C06262=1185.996,260.499,-65.373,-177.131,7.222,148.520
C06263=1185.992,260.748,-65.401,-177.128,7.225,148.520
C06264=1185.988,260.996,-65.428,-177.126,7.227,148.520
C06265=1185.983,261.244,-65.456,-177.124,7.230,148.520
C06266=1185.979,261.492,-65.483,-177.120,7.232,148.519
C06267=1185.975,261.741,-65.511,-177.118,7.235,148.519
C06268=1185.970,261.989,-65.539,-177.115,7.238,148.519
C06269=1185.966,262.263,-65.569,-177.113,7.241,148.519
C06270=1185.960,262.535,-65.600,-177.110,7.243,148.519
C06271=1185.955,262.809,-65.629,-177.107,7.246,148.519
C06272=1185.951,263.081,-65.659,-177.104,7.249,148.519
C06273=1185.946,263.330,-65.688,-177.101,7.251,148.519
C06274=1185.942,263.578,-65.716,-177.099,7.254,148.518
C06275=1185.937,263.827,-65.743,-177.097,7.256,148.518
C06276=1185.933,264.075,-65.771,-177.094,7.259,148.518
C06277=1185.929,264.324,-65.798,-177.092,7.261,148.518
C06278=1185.925,264.572,-65.826,-177.088,7.264,148.518
C06279=1185.920,264.821,-65.855,-177.086,7.267,148.518
C06280=1185.916,265.069,-65.882,-177.084,7.269,148.518
C06281=1185.911,265.317,-65.909,-177.081,7.272,148.518
C06282=1185.907,265.566,-65.937,-177.079,7.274,148.518
C06283=1185.903,265.814,-65.965,-177.075,7.277,148.517
C06284=1185.898,266.062,-65.993,-177.073,7.280,148.517
C06285=1185.894,266.311,-66.021,-177.071,7.282,148.517
C06286=1185.889,266.559,-66.048,-177.068,7.285,148.517
C06287=1185.886,266.808,-66.076,-177.065,7.288,148.517
C06288=1185.880,267.056,-66.105,-177.063,7.290,148.517
C06289=1185.876,267.304,-66.132,-177.060,7.293,148.517
C06290=1185.872,267.552,-66.161,-177.058,7.295,148.517
C06291=1185.867,267.801,-66.188,-177.055,7.298,148.517
C06292=1185.863,268.050,-66.216,-177.052,7.301,148.517
C06293=1185.859,268.298,-66.244,-177.050,7.303,148.517
C06294=1185.855,268.546,-66.272,-177.047,7.306,148.516
C06295=1185.850,268.794,-66.301,-177.045,7.308,148.516
C06296=1185.845,269.043,-66.328,-177.042,7.311,148.516
C06297=1185.842,269.292,-66.356,-177.039,7.314,148.516
C06298=1185.837,269.540,-66.384,-177.037,7.316,148.516
C06299=1185.833,269.788,-66.412,-177.034,7.319,148.516
C06300=1185.828,270.037,-66.441,-177.031,7.322,148.516
C06301=1185.824,270.285,-66.469,-177.029,7.324,148.516
C06302=1185.820,270.533,-66.497,-177.026,7.327,148.516
C06303=1185.815,270.782,-66.525,-177.024,7.330,148.516
C06304=1185.811,271.030,-66.553,-177.021,7.332,148.516
C06305=1185.807,271.278,-66.581,-177.019,7.335,148.516
C06306=1185.802,271.526,-66.610,-177.016,7.337,148.515
C06307=1185.798,271.775,-66.638,-177.013,7.340,148.515
C06308=1185.793,272.023,-66.666,-177.011,7.343,148.515
C06309=1185.789,272.272,-66.694,-177.008,7.345,148.515
C06310=1185.784,272.520,-66.723,-177.006,7.348,148.515
C06311=1185.780,272.769,-66.751,-177.003,7.351,148.515
C06312=1185.775,273.017,-66.779,-177.001,7.353,148.515
C06313=1185.772,273.265,-66.807,-176.998,7.356,148.515
C06314=1185.767,273.513,-66.835,-176.995,7.359,148.515
C06315=1185.763,273.762,-66.864,-176.993,7.361,148.514
C06316=1185.758,274.010,-66.892,-176.990,7.364,148.514
C06317=1185.754,274.259,-66.920,-176.987,7.367,148.514
C06318=1185.750,274.507,-66.949,-176.985,7.369,148.514
C06319=1185.745,274.756,-66.977,-176.982,7.372,148.514
C06320=1185.742,275.004,-67.006,-176.980,7.375,148.514
C06321=1185.737,275.252,-67.034,-176.978,7.377,148.514
C06322=1185.732,275.501,-67.063,-176.975,7.380,148.514
C06323=1185.728,275.749,-67.091,-176.972,7.383,148.514
C06324=1185.723,275.997,-67.119,-176.969,7.385,148.514
C06325=1185.720,276.245,-67.148,-176.967,7.388,148.514
C06326=1185.715,276.494,-67.177,-176.964,7.391,148.514
C06327=1185.711,276.742,-67.205,-176.962,7.393,148.514
C06328=1185.706,276.991,-67.234,-176.959,7.396,148.514
C06329=1185.702,277.238,-67.262,-176.956,7.399,148.514
C06330=1185.698,277.487,-67.291,-176.954,7.401,148.513
C06331=1185.693,277.735,-67.319,-176.951,7.404,148.513
C06332=1185.689,277.984,-67.347,-176.949,7.407,148.513
C06333=1185.685,278.232,-67.377,-176.947,7.410,148.513
C06334=1185.680,278.480,-67.405,-176.944,7.413,148.513
C06335=1185.676,278.729,-67.433,-176.941,7.415,148.513
C06336=1185.672,278.977,-67.463,-176.939,7.417,148.513
C06337=1185.667,279.225,-67.491,-176.936,7.420,148.513
C06338=1185.663,279.473,-67.520,-176.933,7.423,148.513
C06339=1185.659,279.722,-67.549,-176.930,7.426,148.513
C06340=1185.654,279.970,-67.577,-176.928,7.429,148.513
C06341=1185.650,280.218,-67.606,-176.925,7.432,148.513
C06342=1185.646,280.467,-67.635,-176.923,7.435,148.513
C06343=1185.641,280.715,-67.664,-176.921,7.437,148.513
C06344=1185.637,280.963,-67.692,-176.918,7.440,148.513
C06345=1185.633,281.212,-67.721,-176.915,7.443,148.513
C06346=1185.628,281.460,-67.750,-176.913,7.445,148.512
C06347=1185.624,281.708,-67.779,-176.910,7.448,148.512
C06348=1185.620,281.957,-67.807,-176.908,7.451,148.512
C06349=1185.616,282.205,-67.837,-176.905,7.454,148.512
C06350=1185.611,282.453,-67.865,-176.903,7.456,148.512
C06351=1185.607,282.701,-67.895,-176.900,7.459,148.512
C06352=1185.603,282.950,-67.923,-176.897,7.462,148.512
C06353=1185.598,283.198,-67.952,-176.895,7.464,148.512
C06354=1185.594,283.447,-67.981,-176.892,7.467,148.512
C06355=1185.589,283.695,-68.010,-176.890,7.470,148.512
C06356=1185.585,283.943,-68.039,-176.887,7.473,148.512
C06357=1185.580,284.191,-68.068,-176.885,7.475,148.512
C06358=1185.577,284.439,-68.097,-176.882,7.478,148.512
C06359=1185.572,284.688,-68.125,-176.879,7.481,148.512
C06360=1185.568,284.936,-68.155,-176.877,7.483,148.512
C06361=1185.564,285.185,-68.184,-176.874,7.486,148.512
C06362=1185.559,285.433,-68.213,-176.871,7.489,148.512
C06363=1185.555,285.681,-68.242,-176.869,7.492,148.512
C06364=1185.550,285.929,-68.272,-176.866,7.494,148.511
C06365=1185.547,286.177,-68.300,-176.864,7.498,148.512
C06366=1185.542,286.425,-68.329,-176.861,7.501,148.512
C06367=1185.538,286.674,-68.358,-176.859,7.504,148.512
C06368=1185.534,286.922,-68.388,-176.857,7.506,148.511
C06369=1185.529,287.170,-68.417,-176.854,7.509,148.511
C06370=1185.525,287.419,-68.446,-176.851,7.512,148.511
C06371=1185.521,287.667,-68.475,-176.848,7.515,148.511
C06372=1185.516,287.915,-68.504,-176.846,7.517,148.511
C06373=1185.512,288.190,-68.536,-176.843,7.520,148.511
C06374=1185.507,288.464,-68.569,-176.840,7.523,148.511
C06375=1185.502,288.739,-68.601,-176.837,7.526,148.511
C06376=1185.497,289.013,-68.634,-176.834,7.529,148.511
C06377=1185.493,289.262,-68.663,-176.832,7.532,148.511
C06378=1185.488,289.510,-68.693,-176.829,7.535,148.511
C06379=1185.484,289.759,-68.722,-176.827,7.538,148.511
C06380=1185.480,290.007,-68.751,-176.824,7.541,148.511
C06381=1185.476,290.255,-68.781,-176.821,7.544,148.511
C06382=1185.471,290.503,-68.810,-176.820,7.546,148.511
C06383=1185.467,290.751,-68.839,-176.817,7.549,148.511
C06384=1185.463,290.999,-68.869,-176.814,7.552,148.511
C06385=1185.459,291.248,-68.898,-176.811,7.555,148.511
C06386=1185.454,291.496,-68.928,-176.809,7.557,148.511
C06387=1185.450,291.744,-68.957,-176.807,7.560,148.511
C06388=1185.446,291.992,-68.987,-176.804,7.563,148.511
C06389=1185.442,292.241,-69.016,-176.801,7.566,148.511
C06390=1185.437,292.489,-69.046,-176.799,7.568,148.511
C06391=1185.433,292.737,-69.076,-176.796,7.571,148.511
C06392=1185.429,292.986,-69.105,-176.794,7.574,148.511
C06393=1185.424,293.234,-69.135,-176.791,7.577,148.511
C06394=1185.420,293.482,-69.164,-176.788,7.580,148.511
C06395=1185.416,293.729,-69.194,-176.786,7.583,148.510
C06396=1185.411,293.977,-69.223,-176.783,7.586,148.510
C06397=1185.407,294.226,-69.253,-176.781,7.589,148.511
C06398=1185.402,294.474,-69.283,-176.778,7.592,148.511
C06399=1185.398,294.723,-69.312,-176.776,7.594,148.511
C06400=1185.394,294.971,-69.342,-176.773,7.597,148.511
C06401=1185.390,295.219,-69.371,-176.771,7.600,148.511
C06402=1185.386,295.467,-69.401,-176.768,7.603,148.510
C06403=1185.381,295.715,-69.431,-176.765,7.606,148.510
C06404=1185.377,295.964,-69.461,-176.763,7.608,148.510
C06405=1185.373,296.212,-69.490,-176.760,7.611,148.510
C06406=1185.369,296.460,-69.520,-176.758,7.614,148.510
C06407=1185.365,296.708,-69.550,-176.755,7.617,148.511
C06408=1185.360,296.956,-69.580,-176.753,7.620,148.510
C06409=1185.356,297.205,-69.609,-176.750,7.623,148.510
C06410=1185.352,297.452,-69.640,-176.748,7.626,148.510
C06411=1185.347,297.701,-69.670,-176.745,7.629,148.510
C06412=1185.343,297.949,-69.699,-176.742,7.632,148.510
C06413=1185.339,298.197,-69.729,-176.740,7.635,148.510
C06414=1185.335,298.445,-69.759,-176.737,7.637,148.510
C06415=1185.330,298.693,-69.789,-176.735,7.640,148.510
C06416=1185.326,298.942,-69.819,-176.733,7.643,148.510
C06417=1185.322,299.190,-69.849,-176.730,7.646,148.510
C06418=1185.318,299.438,-69.879,-176.727,7.649,148.510
C06419=1185.313,299.686,-69.909,-176.725,7.651,148.510
C06420=1185.309,299.934,-69.939,-176.722,7.654,148.510
C06421=1185.305,300.183,-69.969,-176.719,7.657,148.510
C06422=1185.300,300.431,-69.999,-176.717,7.661,148.510
C06423=1185.296,300.679,-70.029,-176.715,7.664,148.510
C06424=1185.292,300.927,-70.059,-176.712,7.666,148.510
C06425=1185.288,301.175,-70.089,-176.710,7.669,148.510
C06426=1185.283,301.423,-70.119,-176.707,7.672,148.510
C06427=1185.279,301.671,-70.149,-176.704,7.675,148.510
C06428=1185.275,301.920,-70.180,-176.701,7.678,148.510
C06429=1185.271,302.168,-70.210,-176.700,7.680,148.510
C06430=1185.267,302.416,-70.240,-176.697,7.683,148.510
C06431=1185.262,302.664,-70.270,-176.694,7.686,148.510
C06432=1185.258,302.912,-70.300,-176.692,7.689,148.510
C06433=1185.253,303.160,-70.330,-176.689,7.692,148.510
C06434=1185.249,303.408,-70.360,-176.687,7.696,148.511
C06435=1185.245,303.656,-70.391,-176.685,7.698,148.510
C06436=1185.241,303.905,-70.421,-176.682,7.701,148.510
C06437=1185.236,304.153,-70.452,-176.679,7.704,148.510
C06438=1185.233,304.401,-70.482,-176.676,7.707,148.510
C06439=1185.228,304.649,-70.512,-176.674,7.710,148.511
C06440=1185.224,304.897,-70.542,-176.671,7.713,148.511
C06441=1185.219,305.145,-70.573,-176.669,7.715,148.511
C06442=1185.216,305.394,-70.603,-176.667,7.718,148.511
C06443=1185.211,305.642,-70.633,-176.664,7.721,148.511
C06444=1185.206,305.890,-70.664,-176.662,7.724,148.511
C06445=1185.202,306.137,-70.694,-176.659,7.727,148.511
C06446=1185.198,306.386,-70.724,-176.656,7.730,148.511
C06447=1185.194,306.634,-70.755,-176.654,7.733,148.511
C06448=1185.190,306.882,-70.786,-176.651,7.736,148.511
C06449=1185.186,307.130,-70.816,-176.649,7.739,148.511
C06450=1185.181,307.378,-70.847,-176.646,7.742,148.511
C06451=1185.176,307.626,-70.877,-176.644,7.745,148.511
C06452=1185.173,307.875,-70.907,-176.641,7.748,148.511
C06453=1185.168,308.123,-70.938,-176.639,7.750,148.511
C06454=1185.164,308.371,-70.969,-176.636,7.753,148.511
C06455=1185.160,308.618,-70.999,-176.634,7.756,148.511
C06456=1185.156,308.867,-71.030,-176.631,7.759,148.511
C06457=1185.151,309.115,-71.061,-176.629,7.763,148.511
C06458=1185.147,309.363,-71.091,-176.626,7.766,148.511
C06459=1185.143,309.611,-71.122,-176.623,7.769,148.511
C06460=1185.138,309.860,-71.152,-176.621,7.771,148.511
C06461=1185.135,310.107,-71.182,-176.619,7.774,148.511
C06462=1185.130,310.355,-71.213,-176.616,7.777,148.511
C06463=1185.125,310.603,-71.244,-176.614,7.780,148.511
C06464=1185.122,310.852,-71.274,-176.611,7.784,148.511
C06465=1185.117,311.100,-71.305,-176.609,7.787,148.511
C06466=1185.113,311.348,-71.336,-176.606,7.790,148.511
C06467=1185.109,311.596,-71.368,-176.604,7.792,148.511
C06468=1185.105,311.843,-71.398,-176.601,7.795,148.511
C06469=1185.101,312.091,-71.429,-176.599,7.798,148.511
C06470=1185.097,312.340,-71.460,-176.596,7.801,148.511
C06471=1185.092,312.588,-71.491,-176.594,7.804,148.512
C06472=1185.088,312.836,-71.521,-176.591,7.807,148.512
C06473=1185.084,313.084,-71.552,-176.588,7.810,148.512
C06474=1185.080,313.332,-71.583,-176.587,7.813,148.512
C06475=1185.075,313.580,-71.613,-176.584,7.816,148.512
C06476=1185.071,313.829,-71.645,-176.581,7.819,148.512
C06477=1185.066,314.105,-71.679,-176.579,7.822,148.512
C06478=1185.062,314.381,-71.714,-176.576,7.826,148.512
C06479=1185.057,314.658,-71.749,-176.573,7.829,148.512
C06480=1185.052,314.934,-71.782,-176.570,7.832,148.512
C06481=1185.048,315.183,-71.813,-176.568,7.835,148.512
C06482=1185.044,315.430,-71.845,-176.565,7.838,148.512
C06483=1185.040,315.679,-71.876,-176.563,7.841,148.512
C06484=1185.036,315.927,-71.906,-176.560,7.845,148.512
C06485=1185.031,316.174,-71.938,-176.558,7.848,148.512
C06486=1185.027,316.423,-71.969,-176.555,7.851,148.512
C06487=1185.023,316.671,-72.000,-176.553,7.854,148.512
C06488=1185.019,316.919,-72.031,-176.551,7.856,148.512
C06489=1185.014,317.167,-72.062,-176.548,7.859,148.512
C06490=1185.010,317.415,-72.093,-176.546,7.863,148.513
C06491=1185.006,317.663,-72.124,-176.543,7.866,148.513
C06492=1185.002,317.911,-72.156,-176.541,7.869,148.513
C06493=1184.998,318.159,-72.187,-176.538,7.872,148.513
C06494=1184.993,318.407,-72.218,-176.535,7.875,148.513
C06495=1184.989,318.655,-72.249,-176.533,7.878,148.513
C06496=1184.985,318.903,-72.280,-176.531,7.880,148.513
C06497=1184.981,319.151,-72.312,-176.528,7.884,148.513
C06498=1184.976,319.399,-72.343,-176.526,7.887,148.513
C06499=1184.973,319.647,-72.375,-176.523,7.890,148.513
C06500=1184.968,319.895,-72.405,-176.521,7.893,148.513
C06501=1184.964,320.143,-72.437,-176.518,7.896,148.513
C06502=1184.960,320.391,-72.468,-176.516,7.899,148.514
C06503=1184.956,320.639,-72.500,-176.513,7.902,148.514
C06504=1184.951,320.887,-72.531,-176.510,7.905,148.514
C06505=1184.948,321.135,-72.562,-176.508,7.909,148.514
C06506=1184.943,321.383,-72.594,-176.506,7.911,148.514
C06507=1184.939,321.631,-72.625,-176.504,7.914,148.514
C06508=1184.935,321.879,-72.656,-176.501,7.917,148.514
C06509=1184.931,322.127,-72.688,-176.499,7.920,148.514
C06510=1184.927,322.375,-72.719,-176.496,7.923,148.514
C06511=1184.923,322.623,-72.751,-176.494,7.927,148.514
C06512=1184.918,322.871,-72.782,-176.491,7.930,148.514
C06513=1184.914,323.119,-72.814,-176.488,7.933,148.514
C06514=1184.909,323.367,-72.845,-176.486,7.936,148.514
C06515=1184.906,323.615,-72.877,-176.483,7.939,148.514
C06516=1184.901,323.862,-72.908,-176.482,7.942,148.515
C06517=1184.898,324.110,-72.940,-176.479,7.945,148.515
C06518=1184.894,324.359,-72.971,-176.477,7.948,148.515
C06519=1184.889,324.606,-73.003,-176.474,7.951,148.515
C06520=1184.885,324.855,-73.035,-176.472,7.954,148.515
C06521=1184.880,325.103,-73.066,-176.469,7.957,148.515
C06522=1184.876,325.351,-73.098,-176.467,7.961,148.515
C06523=1184.873,325.599,-73.130,-176.464,7.964,148.515
C06524=1184.868,325.846,-73.161,-176.462,7.967,148.515
C06525=1184.864,326.094,-73.193,-176.459,7.970,148.515
C06526=1184.859,326.342,-73.224,-176.457,7.973,148.516
C06527=1184.856,326.590,-73.256,-176.455,7.975,148.516
C06528=1184.852,326.838,-73.288,-176.453,7.979,148.516
C06529=1184.847,327.086,-73.320,-176.450,7.982,148.516
C06530=1184.843,327.334,-73.352,-176.448,7.985,148.516
C06531=1184.839,327.581,-73.383,-176.445,7.988,148.516
C06532=1184.835,327.829,-73.415,-176.443,7.991,148.516
C06533=1184.831,328.078,-73.448,-176.440,7.995,148.516
C06534=1184.826,328.326,-73.478,-176.438,7.998,148.516
C06535=1184.822,328.574,-73.510,-176.435,8.001,148.517
C06536=1184.818,328.822,-73.543,-176.433,8.004,148.517
C06537=1184.814,329.069,-73.574,-176.430,8.007,148.517
C06538=1184.810,329.317,-73.606,-176.428,8.011,148.517
C06539=1184.806,329.566,-73.638,-176.425,8.014,148.517
C06540=1184.801,329.813,-73.670,-176.424,8.016,148.517
C06541=1184.798,330.061,-73.702,-176.421,8.019,148.517
C06542=1184.793,330.310,-73.734,-176.419,8.022,148.517
C06543=1184.789,330.557,-73.766,-176.417,8.026,148.518
C06544=1184.784,330.805,-73.798,-176.414,8.029,148.518
C06545=1184.781,331.053,-73.830,-176.412,8.032,148.518
C06546=1184.777,331.300,-73.862,-176.409,8.035,148.518
C06547=1184.772,331.548,-73.895,-176.407,8.038,148.518
C06548=1184.768,331.796,-73.926,-176.404,8.042,148.518
C06549=1184.764,332.045,-73.959,-176.402,8.045,148.518
C06550=1184.760,332.292,-73.990,-176.399,8.048,148.518
C06551=1184.756,332.540,-74.022,-176.397,8.051,148.519
C06552=1184.752,332.788,-74.055,-176.394,8.054,148.519
C06553=1184.748,333.037,-74.087,-176.392,8.058,148.519
C06554=1184.743,333.284,-74.119,-176.390,8.060,148.519
C06555=1184.739,333.532,-74.151,-176.388,8.063,148.519
C06556=1184.735,333.780,-74.184,-176.386,8.066,148.519
C06557=1184.731,334.028,-74.215,-176.383,8.070,148.519
C06558=1184.726,334.276,-74.247,-176.381,8.073,148.519
C06559=1184.723,334.523,-74.280,-176.378,8.076,148.520
C06560=1184.718,334.771,-74.312,-176.376,8.079,148.520
C06561=1184.715,335.019,-74.344,-176.374,8.083,148.520
C06562=1184.710,335.266,-74.377,-176.371,8.086,148.520
C06563=1184.706,335.514,-74.409,-176.369,8.089,148.520
C06564=1184.702,335.763,-74.441,-176.367,8.092,148.521
C06565=1184.698,336.011,-74.473,-176.364,8.095,148.521
C06566=1184.694,336.259,-74.506,-176.362,8.099,148.521
C06567=1184.689,336.506,-74.538,-176.359,8.102,148.521
C06568=1184.686,336.754,-74.571,-176.357,8.105,148.521
C06569=1184.681,337.002,-74.603,-176.354,8.108,148.521
C06570=1184.677,337.250,-74.635,-176.352,8.112,148.521
C06571=1184.673,337.498,-74.668,-176.350,8.115,148.522
C06572=1184.669,337.746,-74.701,-176.348,8.117,148.522
C06573=1184.665,337.993,-74.733,-176.345,8.120,148.522
C06574=1184.660,338.241,-74.766,-176.343,8.124,148.522
C06575=1184.657,338.489,-74.797,-176.341,8.127,148.522
C06576=1184.652,338.737,-74.831,-176.339,8.130,148.522
C06577=1184.648,338.985,-74.863,-176.336,8.134,148.523
C06578=1184.645,339.233,-74.896,-176.334,8.137,148.523
C06579=1184.640,339.481,-74.928,-176.331,8.140,148.523
C06580=1184.635,339.728,-74.961,-176.329,8.143,148.523
C06581=1184.632,340.007,-74.998,-176.326,8.148,148.523
C06582=1184.627,340.286,-75.034,-176.324,8.151,148.524
C06583=1184.622,340.565,-75.071,-176.322,8.154,148.524
C06584=1184.617,340.844,-75.107,-176.319,8.158,148.524
C06585=1184.613,341.092,-75.140,-176.316,8.161,148.524
C06586=1184.609,341.340,-75.173,-176.314,8.165,148.524
C06587=1184.605,341.587,-75.205,-176.312,8.168,148.524
C06588=1184.601,341.835,-75.239,-176.310,8.171,148.525
C06589=1184.597,342.084,-75.271,-176.307,8.175,148.525
C06590=1184.592,342.331,-75.304,-176.305,8.178,148.525
C06591=1184.588,342.578,-75.336,-176.303,8.181,148.525
C06592=1184.584,342.826,-75.369,-176.300,8.184,148.525
C06593=1184.580,343.074,-75.402,-176.298,8.188,148.526
C06594=1184.576,343.322,-75.435,-176.296,8.191,148.526
C06595=1184.571,343.570,-75.468,-176.294,8.193,148.526
C06596=1184.568,343.818,-75.500,-176.292,8.197,148.526
C06597=1184.564,344.065,-75.533,-176.289,8.200,148.526
C06598=1184.560,344.313,-75.566,-176.287,8.203,148.527
C06599=1184.555,344.561,-75.599,-176.285,8.207,148.527
C06600=1184.551,344.809,-75.632,-176.283,8.210,148.527
C06601=1184.547,345.057,-75.665,-176.280,8.213,148.527
C06602=1184.544,345.304,-75.698,-176.278,8.217,148.527
C06603=1184.539,345.552,-75.731,-176.276,8.220,148.528
C06604=1184.535,345.800,-75.763,-176.274,8.223,148.528
C06605=1184.531,346.048,-75.797,-176.271,8.227,148.528
C06606=1184.527,346.296,-75.830,-176.269,8.230,148.528
C06607=1184.523,346.544,-75.863,-176.267,8.233,148.529
C06608=1184.518,346.791,-75.896,-176.265,8.236,148.529
C06609=1184.514,347.039,-75.929,-176.262,8.240,148.529
C06610=1184.510,347.287,-75.962,-176.260,8.243,148.529
C06611=1184.506,347.534,-75.995,-176.258,8.246,148.529
C06612=1184.502,347.782,-76.029,-176.256,8.250,148.530
C06613=1184.497,348.031,-76.061,-176.253,8.253,148.530
C06614=1184.493,348.278,-76.094,-176.251,8.256,148.530
C06615=1184.490,348.526,-76.127,-176.249,8.260,148.530
C06616=1184.486,348.773,-76.160,-176.247,8.263,148.531
C06617=1184.482,349.021,-76.193,-176.245,8.267,148.531
C06618=1184.477,349.269,-76.226,-176.243,8.270,148.531
C06619=1184.473,349.517,-76.259,-176.240,8.273,148.531
C06620=1184.469,349.764,-76.293,-176.238,8.277,148.532
C06621=1184.465,350.011,-76.326,-176.236,8.280,148.532
C06622=1184.460,350.259,-76.360,-176.233,8.283,148.532
C06623=1184.456,350.507,-76.393,-176.231,8.287,148.532
C06624=1184.452,350.755,-76.427,-176.229,8.290,148.533
C06625=1184.449,351.003,-76.460,-176.227,8.293,148.533
C06626=1184.444,351.251,-76.493,-176.225,8.297,148.533
C06627=1184.440,351.499,-76.526,-176.223,8.300,148.533
C06628=1184.436,351.747,-76.560,-176.220,8.303,148.534
C06629=1184.432,351.994,-76.593,-176.218,8.307,148.534
C06630=1184.428,352.241,-76.627,-176.216,8.310,148.534
C06631=1184.424,352.489,-76.660,-176.214,8.314,148.534
C06632=1184.420,352.737,-76.693,-176.212,8.317,148.535
C06633=1184.416,352.985,-76.726,-176.210,8.320,148.535
C06634=1184.412,353.233,-76.760,-176.208,8.324,148.535
C06635=1184.408,353.480,-76.794,-176.205,8.327,148.536
C06636=1184.404,353.728,-76.827,-176.203,8.331,148.536
C06637=1184.399,353.976,-76.860,-176.201,8.334,148.536
C06638=1184.395,354.224,-76.893,-176.199,8.338,148.536
C06639=1184.391,354.471,-76.927,-176.197,8.341,148.537
C06640=1184.387,354.718,-76.960,-176.195,8.344,148.537
C06641=1184.384,354.967,-76.994,-176.193,8.348,148.537
C06642=1184.379,355.214,-77.028,-176.191,8.351,148.538
C06643=1184.375,355.462,-77.062,-176.188,8.354,148.538
C06644=1184.371,355.710,-77.095,-176.187,8.358,148.538
C06645=1184.367,355.957,-77.129,-176.184,8.361,148.538
C06646=1184.364,356.205,-77.162,-176.182,8.365,148.539
C06647=1184.359,356.453,-77.196,-176.180,8.368,148.539
C06648=1184.355,356.700,-77.230,-176.178,8.372,148.539
C06649=1184.351,356.948,-77.263,-176.176,8.375,148.540
C06650=1184.347,357.195,-77.297,-176.174,8.379,148.540
C06651=1184.343,357.444,-77.331,-176.172,8.382,148.540
C06652=1184.339,357.692,-77.364,-176.170,8.386,148.541
C06653=1184.335,357.939,-77.398,-176.168,8.389,148.541
C06654=1184.331,358.187,-77.431,-176.166,8.392,148.541
C06655=1184.327,358.435,-77.466,-176.163,8.396,148.541
C06656=1184.322,358.682,-77.499,-176.162,8.399,148.542
C06657=1184.319,358.930,-77.533,-176.159,8.403,148.542
C06658=1184.314,359.178,-77.567,-176.158,8.406,148.543
C06659=1184.310,359.425,-77.601,-176.155,8.410,148.543
C06660=1184.307,359.673,-77.635,-176.154,8.413,148.543
C06661=1184.303,359.920,-77.668,-176.151,8.417,148.543
C06662=1184.298,360.168,-77.702,-176.149,8.420,148.544
C06663=1184.294,360.416,-77.736,-176.148,8.423,148.544
C06664=1184.291,360.663,-77.770,-176.146,8.426,148.544
C06665=1184.286,360.911,-77.804,-176.144,8.430,148.545
C06666=1184.282,361.158,-77.837,-176.142,8.433,148.545
C06667=1184.278,361.406,-77.872,-176.140,8.437,148.546
C06668=1184.274,361.654,-77.905,-176.138,8.440,148.546
C06669=1184.270,361.901,-77.939,-176.136,8.444,148.546
C06670=1184.266,362.149,-77.974,-176.134,8.447,148.547
C06671=1184.262,362.397,-78.007,-176.132,8.451,148.547
C06672=1184.258,362.644,-78.041,-176.130,8.454,148.547
C06673=1184.254,362.892,-78.076,-176.128,8.458,148.548
C06674=1184.250,363.139,-78.110,-176.127,8.462,148.548
C06675=1184.245,363.388,-78.144,-176.125,8.465,148.549
C06676=1184.242,363.635,-78.178,-176.123,8.468,148.549
C06677=1184.238,363.883,-78.212,-176.121,8.471,148.549
C06678=1184.234,364.130,-78.246,-176.119,8.475,148.550
C06679=1184.230,364.378,-78.280,-176.118,8.479,148.550
C06680=1184.226,364.626,-78.314,-176.116,8.482,148.551
C06681=1184.222,364.873,-78.348,-176.114,8.486,148.551
C06682=1184.218,365.121,-78.383,-176.112,8.489,148.551
C06683=1184.214,365.368,-78.417,-176.110,8.492,148.552
C06684=1184.210,365.617,-78.451,-176.109,8.496,148.552
C06685=1184.205,365.897,-78.489,-176.106,8.500,148.552
C06686=1184.200,366.179,-78.529,-176.104,8.504,148.553
C06687=1184.196,366.460,-78.568,-176.103,8.507,148.553
C06688=1184.192,366.742,-78.607,-176.101,8.512,148.554
C06689=1184.187,366.989,-78.641,-176.099,8.515,148.554
C06690=1184.184,367.237,-78.675,-176.098,8.518,148.555
C06691=1184.179,367.484,-78.710,-176.096,8.522,148.555
C06692=1184.175,367.732,-78.743,-176.094,8.526,148.556
C06693=1184.171,367.980,-78.778,-176.093,8.528,148.556
C06694=1184.167,368.228,-78.812,-176.091,8.532,148.557
C06695=1184.163,368.475,-78.846,-176.089,8.536,148.557
C06696=1184.159,368.723,-78.881,-176.087,8.539,148.557
C06697=1184.155,368.971,-78.916,-176.086,8.542,148.558
C06698=1184.151,369.218,-78.950,-176.085,8.546,148.558
C06699=1184.147,369.466,-78.984,-176.083,8.550,148.559
C06700=1184.143,369.713,-79.018,-176.081,8.553,148.559
C06701=1184.139,369.961,-79.053,-176.080,8.556,148.560
C06702=1184.135,370.209,-79.088,-176.078,8.560,148.560
C06703=1184.131,370.455,-79.122,-176.077,8.564,148.561
C06704=1184.127,370.703,-79.157,-176.075,8.566,148.561
C06705=1184.123,370.951,-79.191,-176.074,8.570,148.562
C06706=1184.119,371.199,-79.226,-176.072,8.574,148.562
C06707=1184.115,371.446,-79.260,-176.071,8.577,148.563
C06708=1184.110,371.694,-79.295,-176.069,8.580,148.563
C06709=1184.107,371.941,-79.329,-176.067,8.584,148.563
C06710=1184.103,372.189,-79.363,-176.067,8.587,148.564
C06711=1184.099,372.437,-79.398,-176.065,8.591,148.564
C06712=1184.095,372.683,-79.433,-176.064,8.594,148.565
C06713=1184.091,372.931,-79.468,-176.062,8.597,148.565
C06714=1184.087,373.179,-79.502,-176.060,8.601,148.566
C06715=1184.083,373.427,-79.536,-176.059,8.604,148.566
C06716=1184.079,373.674,-79.571,-176.058,8.608,148.567
C06717=1184.075,373.922,-79.606,-176.057,8.611,148.568
C06718=1184.070,374.169,-79.641,-176.055,8.615,148.568
C06719=1184.067,374.417,-79.675,-176.054,8.618,148.569
C06720=1184.063,374.664,-79.710,-176.052,8.621,148.569
C06721=1184.059,374.912,-79.744,-176.052,8.624,148.570
C06722=1184.054,375.159,-79.780,-176.050,8.628,148.570
C06723=1184.051,375.407,-79.814,-176.049,8.631,148.571
C06724=1184.047,375.654,-79.848,-176.048,8.635,148.571
C06725=1184.043,375.902,-79.884,-176.046,8.638,148.572
C06726=1184.039,376.150,-79.919,-176.045,8.642,148.572
C06727=1184.034,376.397,-79.953,-176.044,8.644,148.573
C06728=1184.032,376.645,-79.988,-176.043,8.648,148.573
C06729=1184.027,376.892,-80.022,-176.042,8.652,148.574
C06730=1184.023,377.140,-80.057,-176.040,8.654,148.574
C06731=1184.019,377.387,-80.093,-176.039,8.658,148.575
C06732=1184.015,377.635,-80.127,-176.038,8.661,148.575
C06733=1184.011,377.882,-80.161,-176.037,8.664,148.576
C06734=1184.007,378.130,-80.197,-176.035,8.668,148.576
C06735=1184.003,378.378,-80.232,-176.035,8.671,148.577
C06736=1183.999,378.625,-80.266,-176.034,8.674,148.578
C06737=1183.995,378.873,-80.302,-176.032,8.678,148.578
C06738=1183.990,379.120,-80.336,-176.031,8.681,148.579
C06739=1183.987,379.368,-80.372,-176.030,8.684,148.579
C06740=1183.983,379.615,-80.405,-176.030,8.687,148.580
C06741=1183.979,379.862,-80.441,-176.028,8.691,148.580
C06742=1183.975,380.110,-80.476,-176.027,8.694,148.581
C06743=1183.971,380.357,-80.511,-176.027,8.697,148.582
C06744=1183.967,380.605,-80.546,-176.026,8.700,148.582
C06745=1183.963,380.853,-80.580,-176.024,8.704,148.583
C06746=1183.959,381.100,-80.616,-176.023,8.707,148.583
C06747=1183.955,381.348,-80.651,-176.022,8.710,148.584
C06748=1183.951,381.595,-80.686,-176.021,8.713,148.584
C06749=1183.947,381.843,-80.721,-176.021,8.716,148.585
C06750=1183.942,382.090,-80.756,-176.020,8.719,148.586
C06751=1183.940,382.337,-80.791,-176.019,8.723,148.586
C06752=1183.936,382.585,-80.826,-176.018,8.726,148.587
C06753=1183.931,382.832,-80.861,-176.017,8.730,148.587
C06754=1183.927,383.080,-80.896,-176.016,8.733,148.588
C06755=1183.924,383.328,-80.931,-176.015,8.736,148.588
C06756=1183.919,383.575,-80.966,-176.014,8.739,148.589
C06757=1183.915,383.823,-81.001,-176.014,8.742,148.590
C06758=1183.911,384.070,-81.036,-176.013,8.745,148.590
C06759=1183.907,384.318,-81.071,-176.012,8.748,148.591
C06760=1183.904,384.565,-81.107,-176.012,8.752,148.592
C06761=1183.899,384.813,-81.141,-176.011,8.755,148.592
C06762=1183.895,385.060,-81.177,-176.011,8.757,148.593
C06763=1183.892,385.308,-81.212,-176.010,8.760,148.593
C06764=1183.887,385.555,-81.247,-176.009,8.763,148.594
C06765=1183.883,385.803,-81.282,-176.008,8.766,148.594
C06766=1183.880,386.050,-81.318,-176.008,8.770,148.595
C06767=1183.875,386.297,-81.352,-176.007,8.773,148.596
C06768=1183.871,386.545,-81.388,-176.006,8.776,148.596
C06769=1183.868,386.792,-81.424,-176.006,8.778,148.597
C06770=1183.863,387.040,-81.458,-176.005,8.781,148.597
C06771=1183.860,387.287,-81.494,-176.005,8.785,148.598
C06772=1183.856,387.535,-81.529,-176.004,8.788,148.599
C06773=1183.851,387.782,-81.564,-176.004,8.790,148.599
C06774=1183.848,388.030,-81.599,-176.003,8.793,148.600
C06775=1183.844,388.277,-81.635,-176.002,8.796,148.601
C06776=1183.839,388.525,-81.669,-176.002,8.799,148.601
C06777=1183.836,388.772,-81.705,-176.001,8.802,148.602
C06778=1183.831,389.020,-81.741,-176.001,8.805,148.603
C06779=1183.828,389.268,-81.776,-176.001,8.807,148.603
C06780=1183.823,389.515,-81.811,-176.000,8.810,148.604
C06781=1183.820,389.762,-81.846,-175.999,8.814,148.605
C06782=1183.816,390.010,-81.882,-175.999,8.816,148.605
C06783=1183.812,390.257,-81.917,-175.998,8.819,148.606
C06784=1183.808,390.504,-81.953,-175.999,8.822,148.606
C06785=1183.804,390.752,-81.987,-175.998,8.825,148.607
C06786=1183.800,391.000,-82.023,-175.998,8.827,148.607
C06787=1183.796,391.247,-82.058,-175.997,8.831,148.608
C06788=1183.792,391.494,-82.094,-175.997,8.833,148.609
C06789=1183.788,391.778,-82.134,-175.996,8.836,148.610
C06790=1183.782,392.062,-82.175,-175.996,8.840,148.610
C06791=1183.778,392.347,-82.216,-175.995,8.843,148.611
C06792=1183.774,392.630,-82.256,-175.995,8.846,148.612
C06793=1183.770,392.877,-82.292,-175.995,8.849,148.612
C06794=1183.766,393.125,-82.326,-175.995,8.851,148.613
C06795=1183.762,393.372,-82.362,-175.994,8.854,148.614
C06796=1183.758,393.620,-82.398,-175.994,8.857,148.614
C06797=1183.755,393.867,-82.433,-175.994,8.859,148.615
C06798=1183.750,394.114,-82.469,-175.994,8.862,148.616
C06799=1183.746,394.362,-82.504,-175.993,8.865,148.616
C06800=1183.742,394.609,-82.540,-175.993,8.867,148.617
C06801=1183.739,394.857,-82.575,-175.993,8.870,148.617
C06802=1183.734,395.104,-82.610,-175.992,8.872,148.618
C06803=1183.730,395.352,-82.646,-175.993,8.875,148.619
C06804=1183.726,395.600,-82.682,-175.992,8.878,148.619
C06805=1183.722,395.847,-82.717,-175.992,8.881,148.620
C06806=1183.718,396.094,-82.752,-175.992,8.883,148.620
C06807=1183.715,396.341,-82.788,-175.992,8.886,148.621
C06808=1183.711,396.589,-82.823,-175.992,8.888,148.622
C06809=1183.707,396.836,-82.859,-175.991,8.891,148.622
C06810=1183.702,397.084,-82.895,-175.991,8.893,148.623
C06811=1183.699,397.331,-82.930,-175.991,8.896,148.624
C06812=1183.695,397.579,-82.966,-175.991,8.898,148.624
C06813=1183.691,397.826,-83.001,-175.991,8.901,148.625
C06814=1183.687,398.073,-83.037,-175.991,8.903,148.625
C06815=1183.682,398.321,-83.072,-175.990,8.906,148.626
C06816=1183.679,398.569,-83.108,-175.990,8.909,148.627
C06817=1183.675,398.816,-83.143,-175.990,8.911,148.627
C06818=1183.671,399.064,-83.179,-175.990,8.914,148.628
C06819=1183.667,399.311,-83.214,-175.990,8.916,148.629
C06820=1183.663,399.558,-83.250,-175.990,8.918,148.629
C06821=1183.659,399.806,-83.286,-175.990,8.921,148.630
C06822=1183.655,400.053,-83.321,-175.990,8.923,148.630
C06823=1183.652,400.301,-83.357,-175.990,8.926,148.631
C06824=1183.647,400.548,-83.392,-175.989,8.928,148.632
C06825=1183.643,400.796,-83.428,-175.990,8.930,148.632
C06826=1183.639,401.043,-83.464,-175.989,8.933,148.633
C06827=1183.636,401.291,-83.499,-175.989,8.935,148.633
C06828=1183.631,401.537,-83.534,-175.989,8.937,148.634
C06829=1183.627,401.785,-83.570,-175.989,8.940,148.635
C06830=1183.623,402.033,-83.606,-175.989,8.942,148.635
C06831=1183.620,402.280,-83.642,-175.989,8.945,148.636
C06832=1183.616,402.527,-83.678,-175.989,8.947,148.636
C06833=1183.611,402.774,-83.714,-175.989,8.949,148.637
C06834=1183.608,403.022,-83.749,-175.989,8.952,148.638
C06835=1183.604,403.269,-83.785,-175.989,8.954,148.638
C06836=1183.600,403.517,-83.820,-175.989,8.956,148.639
C06837=1183.596,403.764,-83.856,-175.989,8.958,148.639
C06838=1183.592,404.012,-83.892,-175.989,8.960,148.640
C06839=1183.588,404.259,-83.927,-175.989,8.963,148.641
C06840=1183.584,404.507,-83.963,-175.989,8.965,148.641
C06841=1183.580,404.754,-83.999,-175.989,8.968,148.642
C06842=1183.576,405.002,-84.034,-175.988,8.970,148.642
C06843=1183.573,405.249,-84.070,-175.989,8.972,148.643
C06844=1183.568,405.496,-84.106,-175.989,8.974,148.643
C06845=1183.564,405.744,-84.141,-175.989,8.976,148.644
C06846=1183.561,405.991,-84.177,-175.989,8.979,148.645
C06847=1183.557,406.238,-84.213,-175.989,8.981,148.645
C06848=1183.552,406.486,-84.249,-175.989,8.982,148.646
C06849=1183.549,406.733,-84.285,-175.989,8.985,148.646
C06850=1183.545,406.980,-84.320,-175.989,8.987,148.647
C06851=1183.540,407.228,-84.356,-175.988,8.989,148.647
C06852=1183.536,407.475,-84.392,-175.989,8.992,148.648
C06853=1183.533,407.723,-84.427,-175.989,8.993,148.649
C06854=1183.528,407.971,-84.463,-175.989,8.996,148.649
C06855=1183.525,408.218,-84.500,-175.989,8.998,148.650
C06856=1183.521,408.464,-84.535,-175.989,9.000,148.650
C06857=1183.517,408.712,-84.570,-175.989,9.002,148.651
C06858=1183.513,408.960,-84.606,-175.989,9.004,148.651
C06859=1183.509,409.207,-84.642,-175.989,9.007,148.652
C06860=1183.505,409.455,-84.677,-175.989,9.008,148.653
C06861=1183.501,409.702,-84.714,-175.989,9.011,148.653
C06862=1183.498,409.949,-84.750,-175.989,9.013,148.654
C06863=1183.493,410.196,-84.785,-175.989,9.015,148.654
C06864=1183.489,410.444,-84.821,-175.989,9.017,148.655
C06865=1183.485,410.692,-84.857,-175.989,9.019,148.655
C06866=1183.482,410.939,-84.892,-175.990,9.021,148.656
C06867=1183.478,411.186,-84.929,-175.989,9.023,148.657
C06868=1183.474,411.434,-84.965,-175.989,9.025,148.657
C06869=1183.470,411.681,-85.000,-175.989,9.027,148.657
C06870=1183.465,411.928,-85.036,-175.989,9.029,148.658
C06871=1183.462,412.176,-85.072,-175.989,9.032,148.659
C06872=1183.458,412.423,-85.107,-175.990,9.033,148.659
C06873=1183.454,412.671,-85.144,-175.989,9.035,148.660
C06874=1183.450,412.918,-85.180,-175.990,9.037,148.660
C06875=1183.446,413.166,-85.215,-175.989,9.039,148.661
C06876=1183.442,413.413,-85.251,-175.989,9.041,148.661
C06877=1183.438,413.660,-85.287,-175.990,9.043,148.662
C06878=1183.434,413.907,-85.323,-175.990,9.045,148.662
C06879=1183.430,414.155,-85.359,-175.990,9.047,148.663
C06880=1183.426,414.402,-85.394,-175.990,9.049,148.663
C06881=1183.422,414.650,-85.430,-175.989,9.051,148.664
C06882=1183.419,414.897,-85.467,-175.990,9.053,148.664
C06883=1183.415,415.145,-85.502,-175.989,9.055,148.665
C06884=1183.410,415.392,-85.538,-175.990,9.057,148.666
C06885=1183.407,415.610,-85.570,-175.989,9.059,148.666
C06886=1183.404,415.828,-85.602,-175.990,9.060,148.666
C06887=1183.402,416.045,-85.633,-175.990,9.062,148.667
C06888=1183.400,416.264,-85.664,-175.990,9.064,148.667
C06889=1183.399,416.481,-85.696,-175.990,9.065,148.668
C06890=1183.400,416.699,-85.728,-175.990,9.066,148.668
C06891=1183.401,416.917,-85.758,-175.990,9.069,148.669
C06892=1183.403,417.134,-85.789,-175.989,9.070,148.669
C06893=1182.982,417.135,-85.831,-175.993,9.081,148.673
C06894=1182.980,416.916,-85.799,-175.993,9.079,148.672
C06895=1182.979,416.697,-85.768,-175.993,9.077,148.672
C06896=1182.978,416.478,-85.737,-175.993,9.076,148.671
C06897=1182.979,416.259,-85.705,-175.993,9.074,148.671
C06898=1182.980,416.039,-85.674,-175.993,9.072,148.670
C06899=1182.983,415.820,-85.642,-175.993,9.071,148.670
C06900=1182.986,415.600,-85.610,-175.993,9.070,148.670
C06901=1182.990,415.381,-85.578,-175.993,9.067,148.669
C06902=1182.993,415.133,-85.542,-175.993,9.066,148.669
C06903=1182.997,414.886,-85.507,-175.993,9.064,148.668
C06904=1183.001,414.638,-85.471,-175.992,9.062,148.668
C06905=1183.005,414.391,-85.434,-175.993,9.060,148.667
C06906=1183.009,414.144,-85.399,-175.993,9.057,148.666
C06907=1183.013,413.897,-85.363,-175.993,9.056,148.666
C06908=1183.017,413.649,-85.328,-175.993,9.054,148.665
C06909=1183.020,413.402,-85.291,-175.992,9.052,148.665
C06910=1183.025,413.154,-85.255,-175.993,9.050,148.665
C06911=1183.028,412.907,-85.220,-175.992,9.048,148.664
C06912=1183.033,412.659,-85.183,-175.992,9.046,148.663
C06913=1183.036,412.411,-85.148,-175.993,9.044,148.663
C06914=1183.040,412.165,-85.112,-175.992,9.042,148.662
C06915=1183.045,411.918,-85.076,-175.993,9.040,148.662
C06916=1183.049,411.670,-85.040,-175.992,9.037,148.661
C06917=1183.052,411.423,-85.005,-175.992,9.036,148.661
C06918=1183.057,411.175,-84.969,-175.992,9.034,148.660
C06919=1183.060,410.928,-84.932,-175.992,9.032,148.660
C06920=1183.064,410.680,-84.897,-175.992,9.030,148.659
C06921=1183.069,410.433,-84.861,-175.992,9.027,148.658
C06922=1183.072,410.186,-84.825,-175.992,9.026,148.658
C06923=1183.076,409.938,-84.790,-175.992,9.024,148.657
C06924=1183.080,409.691,-84.753,-175.992,9.021,148.657
C06925=1183.084,409.444,-84.718,-175.992,9.020,148.656
C06926=1183.087,409.196,-84.682,-175.992,9.018,148.656
C06927=1183.092,408.948,-84.646,-175.992,9.015,148.655
C06928=1183.096,408.701,-84.611,-175.992,9.013,148.655
C06929=1183.100,408.454,-84.575,-175.992,9.011,148.654
C06930=1183.104,408.207,-84.538,-175.992,9.009,148.654
C06931=1183.107,407.959,-84.503,-175.992,9.006,148.653
C06932=1183.111,407.712,-84.467,-175.991,9.005,148.652
C06933=1183.115,407.464,-84.432,-175.992,9.003,148.652
C06934=1183.120,407.217,-84.396,-175.992,9.000,148.651
C06935=1183.123,406.970,-84.360,-175.992,8.998,148.651
C06936=1183.127,406.722,-84.325,-175.991,8.996,148.650
C06937=1183.131,406.474,-84.289,-175.991,8.994,148.649
C06938=1183.135,406.227,-84.252,-175.992,8.992,148.649
C06939=1183.138,405.980,-84.217,-175.992,8.989,148.648
C06940=1183.143,405.733,-84.181,-175.992,8.987,148.648
C06941=1183.147,405.485,-84.145,-175.991,8.985,148.647
C06942=1183.151,405.238,-84.110,-175.992,8.983,148.647
C06943=1183.154,404.990,-84.074,-175.991,8.981,148.646
C06944=1183.159,404.742,-84.038,-175.992,8.978,148.645
C06945=1183.163,404.495,-84.003,-175.992,8.976,148.645
C06946=1183.167,404.248,-83.967,-175.992,8.973,148.644
C06947=1183.170,404.001,-83.931,-175.991,8.972,148.644
C06948=1183.175,403.754,-83.895,-175.991,8.969,148.643
C06949=1183.178,403.506,-83.860,-175.992,8.967,148.642
C06950=1183.182,403.259,-83.824,-175.991,8.965,148.642
C06951=1183.187,403.011,-83.788,-175.992,8.962,148.641
C06952=1183.191,402.764,-83.753,-175.992,8.960,148.641
C06953=1183.194,402.516,-83.717,-175.992,8.957,148.640
C06954=1183.198,402.269,-83.682,-175.992,8.955,148.639
C06955=1183.202,402.021,-83.645,-175.992,8.953,148.639
C06956=1183.207,401.774,-83.610,-175.992,8.950,148.638
C06957=1183.210,401.527,-83.575,-175.992,8.949,148.638
C06958=1183.214,401.279,-83.539,-175.992,8.946,148.637
C06959=1183.218,401.031,-83.503,-175.992,8.944,148.637
C06960=1183.222,400.784,-83.467,-175.992,8.942,148.636
C06961=1183.226,400.537,-83.432,-175.992,8.939,148.635
C06962=1183.230,400.290,-83.397,-175.992,8.937,148.635
C06963=1183.234,400.042,-83.361,-175.992,8.934,148.634
C06964=1183.238,399.794,-83.325,-175.992,8.932,148.633
C06965=1183.242,399.547,-83.289,-175.992,8.930,148.633
C06966=1183.246,399.300,-83.254,-175.993,8.927,148.632
C06967=1183.250,399.053,-83.219,-175.993,8.924,148.631
C06968=1183.254,398.805,-83.183,-175.993,8.922,148.631
C06969=1183.258,398.557,-83.147,-175.993,8.919,148.630
C06970=1183.261,398.310,-83.112,-175.993,8.917,148.630
C06971=1183.266,398.063,-83.076,-175.993,8.914,148.629
C06972=1183.269,397.815,-83.041,-175.993,8.912,148.628
C06973=1183.274,397.568,-83.005,-175.993,8.909,148.628
C06974=1183.277,397.320,-82.969,-175.993,8.907,148.627
C06975=1183.281,397.073,-82.934,-175.994,8.904,148.626
C06976=1183.285,396.826,-82.898,-175.994,8.902,148.626
C06977=1183.289,396.578,-82.863,-175.994,8.899,148.625
C06978=1183.293,396.331,-82.827,-175.994,8.897,148.625
C06979=1183.297,396.084,-82.792,-175.994,8.894,148.624
C06980=1183.301,395.836,-82.756,-175.995,8.891,148.623
C06981=1183.305,395.589,-82.720,-175.995,8.889,148.623
C06982=1183.309,395.341,-82.686,-175.995,8.886,148.622
C06983=1183.312,395.093,-82.650,-175.995,8.884,148.622
C06984=1183.317,394.846,-82.614,-175.995,8.881,148.621
C06985=1183.321,394.598,-82.579,-175.996,8.878,148.620
C06986=1183.325,394.351,-82.543,-175.995,8.876,148.620
C06987=1183.328,394.103,-82.508,-175.996,8.873,148.619
C06988=1183.333,393.857,-82.472,-175.996,8.870,148.618
C06989=1183.336,393.609,-82.437,-175.996,8.868,148.618
C06990=1183.341,393.361,-82.401,-175.997,8.865,148.617
C06991=1183.345,393.113,-82.366,-175.997,8.862,148.616
C06992=1183.349,392.866,-82.331,-175.997,8.860,148.616
C06993=1183.353,392.619,-82.295,-175.998,8.856,148.615
C06994=1183.357,392.336,-82.254,-175.998,8.854,148.615
C06995=1183.361,392.051,-82.214,-175.998,8.851,148.614
C06996=1183.366,391.767,-82.173,-175.999,8.847,148.613
C06997=1183.371,391.483,-82.133,-175.999,8.844,148.612
C06998=1183.375,391.236,-82.097,-175.999,8.842,148.612
C06999=1183.378,390.988,-82.061,-176.000,8.839,148.611
C07000=1183.383,390.741,-82.026,-176.000,8.836,148.610
C07001=1183.387,390.493,-81.991,-176.001,8.833,148.610
C07002=1183.390,390.246,-81.956,-176.000,8.830,148.609
C07003=1183.395,389.999,-81.921,-176.001,8.827,148.609
C07004=1183.398,389.751,-81.885,-176.002,8.824,148.608
C07005=1183.402,389.504,-81.850,-176.002,8.822,148.607
C07006=1183.406,389.256,-81.815,-176.003,8.819,148.607
C07007=1183.410,389.009,-81.780,-176.003,8.816,148.606
C07008=1183.415,388.761,-81.743,-176.003,8.813,148.605
C07009=1183.418,388.514,-81.708,-176.004,8.810,148.605
C07010=1183.423,388.266,-81.673,-176.004,8.808,148.604
C07011=1183.426,388.019,-81.638,-176.005,8.804,148.603
C07012=1183.430,387.771,-81.602,-176.006,8.801,148.603
C07013=1183.434,387.525,-81.567,-176.006,8.798,148.602
C07014=1183.438,387.276,-81.532,-176.006,8.795,148.602
C07015=1183.442,387.029,-81.497,-176.007,8.792,148.601
C07016=1183.446,386.782,-81.462,-176.008,8.789,148.600
C07017=1183.450,386.534,-81.427,-176.009,8.786,148.600
C07018=1183.454,386.286,-81.391,-176.009,8.784,148.599
C07019=1183.458,386.039,-81.356,-176.009,8.780,148.599
C07020=1183.462,385.792,-81.321,-176.010,8.777,148.598
C07021=1183.466,385.544,-81.286,-176.011,8.774,148.597
C07022=1183.469,385.297,-81.250,-176.012,8.771,148.597
C07023=1183.474,385.049,-81.216,-176.013,8.768,148.596
C07024=1183.478,384.802,-81.180,-176.013,8.765,148.595
C07025=1183.482,384.555,-81.145,-176.014,8.762,148.595
C07026=1183.486,384.307,-81.110,-176.015,8.758,148.594
C07027=1183.490,384.059,-81.075,-176.015,8.755,148.594
C07028=1183.494,383.812,-81.040,-176.016,8.752,148.593
C07029=1183.498,383.564,-81.004,-176.017,8.749,148.593
C07030=1183.501,383.317,-80.969,-176.018,8.746,148.592
C07031=1183.506,383.069,-80.934,-176.019,8.743,148.591
C07032=1183.510,382.822,-80.899,-176.020,8.740,148.591
C07033=1183.514,382.574,-80.864,-176.020,8.737,148.590
C07034=1183.518,382.327,-80.829,-176.021,8.734,148.590
C07035=1183.522,382.079,-80.794,-176.022,8.731,148.589
C07036=1183.526,381.832,-80.759,-176.023,8.728,148.588
C07037=1183.530,381.585,-80.723,-176.024,8.724,148.588
C07038=1183.533,381.337,-80.689,-176.024,8.721,148.587
C07039=1183.537,381.090,-80.654,-176.026,8.717,148.587
C07040=1183.541,380.842,-80.619,-176.027,8.714,148.586
C07041=1183.545,380.594,-80.584,-176.027,8.711,148.585
C07042=1183.550,380.347,-80.549,-176.028,8.708,148.585
C07043=1183.553,380.099,-80.514,-176.029,8.705,148.584
C07044=1183.558,379.852,-80.479,-176.030,8.701,148.584
C07045=1183.562,379.604,-80.444,-176.031,8.698,148.583
C07046=1183.565,379.356,-80.409,-176.033,8.695,148.583
C07047=1183.570,379.109,-80.374,-176.033,8.692,148.582
C07048=1183.573,378.862,-80.339,-176.035,8.688,148.581
C07049=1183.577,378.614,-80.305,-176.036,8.685,148.581
C07050=1183.581,378.367,-80.269,-176.036,8.682,148.580
C07051=1183.586,378.119,-80.235,-176.038,8.678,148.580
C07052=1183.590,377.871,-80.200,-176.039,8.675,148.579
C07053=1183.593,377.624,-80.164,-176.040,8.672,148.579
C07054=1183.598,377.376,-80.130,-176.041,8.668,148.578
C07055=1183.601,377.129,-80.095,-176.042,8.666,148.578
C07056=1183.605,376.882,-80.061,-176.044,8.662,148.577
C07057=1183.609,376.634,-80.026,-176.045,8.658,148.576
C07058=1183.614,376.387,-79.991,-176.046,8.656,148.576
C07059=1183.618,376.139,-79.956,-176.047,8.652,148.575
C07060=1183.621,375.892,-79.922,-176.048,8.649,148.575
C07061=1183.625,375.644,-79.886,-176.050,8.645,148.574
C07062=1183.630,375.397,-79.852,-176.051,8.642,148.574
C07063=1183.634,375.149,-79.817,-176.052,8.638,148.573
C07064=1183.638,374.900,-79.782,-176.053,8.635,148.573
C07065=1183.641,374.654,-79.748,-176.055,8.631,148.572
C07066=1183.645,374.406,-79.713,-176.056,8.629,148.572
C07067=1183.650,374.158,-79.678,-176.057,8.625,148.571
C07068=1183.654,373.910,-79.643,-176.059,8.622,148.571
C07069=1183.657,373.664,-79.609,-176.060,8.618,148.570
C07070=1183.661,373.416,-79.574,-176.061,8.615,148.570
C07071=1183.666,373.168,-79.540,-176.063,8.611,148.569
C07072=1183.669,372.920,-79.505,-176.064,8.608,148.569
C07073=1183.673,372.673,-79.471,-176.066,8.605,148.568
C07074=1183.677,372.426,-79.435,-176.067,8.601,148.568
C07075=1183.682,372.178,-79.401,-176.068,8.598,148.567
C07076=1183.685,371.930,-79.367,-176.070,8.594,148.567
C07077=1183.689,371.683,-79.332,-176.071,8.591,148.566
C07078=1183.693,371.435,-79.297,-176.073,8.588,148.566
C07079=1183.697,371.188,-79.263,-176.074,8.584,148.565
C07080=1183.702,370.940,-79.229,-176.076,8.580,148.565
C07081=1183.706,370.692,-79.194,-176.077,8.577,148.564
C07082=1183.709,370.446,-79.160,-176.079,8.574,148.564
C07083=1183.713,370.197,-79.125,-176.080,8.570,148.563
C07084=1183.718,369.950,-79.090,-176.082,8.567,148.563
C07085=1183.721,369.702,-79.056,-176.083,8.563,148.563
C07086=1183.726,369.455,-79.022,-176.085,8.560,148.562
C07087=1183.729,369.207,-78.987,-176.087,8.556,148.562
C07088=1183.734,368.960,-78.953,-176.088,8.553,148.561
C07089=1183.738,368.712,-78.918,-176.090,8.549,148.561
C07090=1183.741,368.464,-78.884,-176.091,8.546,148.560
C07091=1183.746,368.217,-78.850,-176.093,8.542,148.560
C07092=1183.749,367.969,-78.815,-176.094,8.539,148.559
C07093=1183.754,367.722,-78.781,-176.096,8.536,148.559
C07094=1183.758,367.474,-78.746,-176.098,8.532,148.559
C07095=1183.761,367.227,-78.712,-176.100,8.529,148.558
C07096=1183.766,366.979,-78.678,-176.101,8.526,148.558
C07097=1183.770,366.731,-78.644,-176.103,8.522,148.557
C07098=1183.774,366.449,-78.605,-176.105,8.518,148.557
C07099=1183.779,366.168,-78.566,-176.107,8.514,148.556
C07100=1183.783,365.887,-78.527,-176.109,8.510,148.556
C07101=1183.788,365.605,-78.488,-176.111,8.506,148.555
C07102=1183.791,365.358,-78.454,-176.112,8.503,148.555
C07103=1183.796,365.110,-78.419,-176.114,8.499,148.554
C07104=1183.800,364.862,-78.386,-176.116,8.496,148.554
C07105=1183.804,364.614,-78.351,-176.118,8.492,148.554
C07106=1183.808,364.367,-78.317,-176.120,8.489,148.553
C07107=1183.813,364.120,-78.283,-176.122,8.485,148.553
C07108=1183.816,363.872,-78.249,-176.124,8.481,148.552
C07109=1183.821,363.624,-78.215,-176.125,8.478,148.552
C07110=1183.824,363.377,-78.181,-176.127,8.475,148.552
C07111=1183.828,363.129,-78.147,-176.129,8.472,148.551
C07112=1183.832,362.882,-78.112,-176.131,8.468,148.551
C07113=1183.836,362.634,-78.079,-176.132,8.464,148.551
C07114=1183.840,362.386,-78.044,-176.135,8.461,148.550
C07115=1183.844,362.139,-78.011,-176.137,8.458,148.550
C07116=1183.849,361.891,-77.977,-176.138,8.454,148.550
C07117=1183.852,361.643,-77.943,-176.141,8.451,148.549
C07118=1183.856,361.396,-77.909,-176.142,8.447,148.549
C07119=1183.861,361.148,-77.875,-176.144,8.443,148.548
C07120=1183.864,360.900,-77.841,-176.146,8.440,148.548
C07121=1183.868,360.653,-77.807,-176.148,8.436,148.548
C07122=1183.873,360.405,-77.773,-176.150,8.433,148.547
C07123=1183.877,360.158,-77.739,-176.152,8.429,148.547
C07124=1183.880,359.909,-77.706,-176.154,8.426,148.547
C07125=1183.885,359.662,-77.671,-176.156,8.423,148.547
C07126=1183.889,359.415,-77.637,-176.158,8.420,148.546
C07127=1183.892,359.166,-77.604,-176.160,8.416,148.546
C07128=1183.897,358.919,-77.569,-176.162,8.413,148.545
C07129=1183.901,358.671,-77.536,-176.164,8.409,148.545
C07130=1183.905,358.424,-77.502,-176.166,8.406,148.545
C07131=1183.909,358.175,-77.468,-176.168,8.403,148.545
C07132=1183.913,357.928,-77.434,-176.170,8.399,148.544
C07133=1183.917,357.680,-77.401,-176.172,8.396,148.544
C07134=1183.921,357.433,-77.367,-176.174,8.392,148.543
C07135=1183.926,357.185,-77.334,-176.176,8.389,148.543
C07136=1183.929,356.937,-77.299,-176.178,8.385,148.543
C07137=1183.933,356.690,-77.266,-176.181,8.381,148.543
C07138=1183.937,356.442,-77.233,-176.183,8.378,148.542
C07139=1183.942,356.195,-77.199,-176.185,8.374,148.542
C07140=1183.946,355.947,-77.165,-176.187,8.371,148.542
C07141=1183.950,355.698,-77.132,-176.189,8.367,148.541
C07142=1183.953,355.451,-77.098,-176.191,8.364,148.541
C07143=1183.957,355.204,-77.065,-176.194,8.360,148.541
C07144=1183.962,354.956,-77.030,-176.196,8.357,148.541
C07145=1183.966,354.708,-76.997,-176.198,8.353,148.540
C07146=1183.970,354.460,-76.964,-176.200,8.350,148.540
C07147=1183.974,354.212,-76.931,-176.202,8.347,148.540
C07148=1183.978,353.965,-76.897,-176.204,8.344,148.539
C07149=1183.982,353.717,-76.864,-176.206,8.340,148.539
C07150=1183.987,353.469,-76.830,-176.208,8.337,148.539
C07151=1183.991,353.222,-76.797,-176.211,8.333,148.539
C07152=1183.995,352.975,-76.763,-176.212,8.330,148.538
C07153=1183.998,352.726,-76.729,-176.215,8.326,148.538
C07154=1184.002,352.478,-76.696,-176.217,8.323,148.538
C07155=1184.006,352.231,-76.663,-176.219,8.320,148.537
C07156=1184.010,351.984,-76.629,-176.222,8.316,148.537
C07157=1184.014,351.736,-76.596,-176.223,8.313,148.537
C07158=1184.019,351.488,-76.563,-176.226,8.309,148.537
C07159=1184.023,351.240,-76.530,-176.228,8.306,148.536
C07160=1184.027,350.993,-76.496,-176.230,8.303,148.536
C07161=1184.032,350.745,-76.463,-176.232,8.299,148.536
C07162=1184.035,350.496,-76.429,-176.235,8.296,148.536
C07163=1184.039,350.248,-76.396,-176.236,8.293,148.535
C07164=1184.044,350.001,-76.363,-176.239,8.289,148.535
C07165=1184.047,349.754,-76.329,-176.241,8.286,148.535
C07166=1184.052,349.506,-76.296,-176.243,8.283,148.535
C07167=1184.056,349.258,-76.263,-176.245,8.279,148.534
C07168=1184.060,349.010,-76.229,-176.248,8.276,148.534
C07169=1184.064,348.763,-76.196,-176.250,8.273,148.534
C07170=1184.068,348.515,-76.163,-176.252,8.269,148.534
C07171=1184.072,348.267,-76.130,-176.254,8.266,148.533
C07172=1184.076,348.019,-76.097,-176.256,8.262,148.533
C07173=1184.081,347.772,-76.064,-176.258,8.260,148.533
C07174=1184.085,347.523,-76.031,-176.260,8.257,148.533
C07175=1184.088,347.276,-75.999,-176.262,8.253,148.533
C07176=1184.092,347.028,-75.966,-176.265,8.250,148.532
C07177=1184.097,346.781,-75.932,-176.267,8.247,148.532
C07178=1184.101,346.533,-75.899,-176.269,8.243,148.532
C07179=1184.105,346.285,-75.866,-176.272,8.240,148.532
C07180=1184.109,346.037,-75.833,-176.274,8.237,148.531
C07181=1184.113,345.790,-75.800,-176.276,8.233,148.531
C07182=1184.117,345.542,-75.767,-176.278,8.230,148.531
C07183=1184.122,345.294,-75.734,-176.281,8.227,148.531
C07184=1184.126,345.046,-75.701,-176.283,8.223,148.531
C07185=1184.129,344.798,-75.668,-176.285,8.220,148.530
C07186=1184.133,344.551,-75.635,-176.287,8.217,148.530
C07187=1184.138,344.303,-75.602,-176.290,8.213,148.530
C07188=1184.142,344.055,-75.570,-176.292,8.210,148.530
C07189=1184.146,343.807,-75.537,-176.294,8.207,148.529
C07190=1184.150,343.559,-75.503,-176.296,8.203,148.529
C07191=1184.154,343.311,-75.470,-176.299,8.200,148.529
C07192=1184.158,343.063,-75.438,-176.301,8.197,148.529
C07193=1184.162,342.816,-75.405,-176.304,8.194,148.529
C07194=1184.166,342.568,-75.372,-176.306,8.191,148.529
C07195=1184.171,342.320,-75.340,-176.308,8.187,148.528
C07196=1184.175,342.072,-75.306,-176.310,8.184,148.528
C07197=1184.179,341.825,-75.274,-176.313,8.181,148.528
C07198=1184.183,341.577,-75.242,-176.315,8.177,148.528
C07199=1184.188,341.329,-75.209,-176.317,8.174,148.527
C07200=1184.192,341.081,-75.176,-176.319,8.171,148.527
C07201=1184.195,340.833,-75.144,-176.322,8.168,148.527
C07202=1184.201,340.554,-75.107,-176.324,8.164,148.527
C07203=1184.205,340.276,-75.070,-176.327,8.160,148.527
C07204=1184.209,339.997,-75.033,-176.329,8.157,148.527
C07205=1184.214,339.717,-74.997,-176.332,8.153,148.526
C07206=1184.218,339.470,-74.964,-176.334,8.149,148.526
C07207=1184.222,339.221,-74.932,-176.337,8.146,148.526
C07208=1184.227,338.974,-74.899,-176.339,8.143,148.526
C07209=1184.231,338.726,-74.867,-176.342,8.140,148.526
C07210=1184.235,338.478,-74.834,-176.343,8.137,148.525
C07211=1184.239,338.230,-74.801,-176.346,8.134,148.525
C07212=1184.243,337.983,-74.769,-176.348,8.131,148.525
C07213=1184.247,337.734,-74.736,-176.351,8.128,148.525
C07214=1184.251,337.488,-74.704,-176.353,8.124,148.525
C07215=1184.256,337.239,-74.672,-176.355,8.121,148.525
C07216=1184.260,336.992,-74.639,-176.358,8.118,148.525
C07217=1184.263,336.744,-74.607,-176.360,8.115,148.524
C07218=1184.268,336.495,-74.574,-176.362,8.111,148.524
C07219=1184.271,336.248,-74.542,-176.365,8.108,148.524
C07220=1184.276,336.000,-74.510,-176.367,8.105,148.524
C07221=1184.281,335.752,-74.477,-176.370,8.102,148.524
C07222=1184.284,335.504,-74.445,-176.372,8.098,148.524
C07223=1184.289,335.256,-74.412,-176.374,8.095,148.523
C07224=1184.292,335.008,-74.380,-176.377,8.092,148.523
C07225=1184.297,334.761,-74.348,-176.379,8.089,148.523
C07226=1184.301,334.513,-74.316,-176.381,8.085,148.523
C07227=1184.305,334.265,-74.283,-176.384,8.082,148.523
C07228=1184.309,334.017,-74.251,-176.386,8.079,148.523
C07229=1184.314,333.769,-74.219,-176.388,8.076,148.522
C07230=1184.317,333.521,-74.187,-176.391,8.073,148.522
C07231=1184.322,333.273,-74.154,-176.393,8.070,148.522
C07232=1184.326,333.025,-74.122,-176.395,8.067,148.522
C07233=1184.331,332.777,-74.090,-176.398,8.064,148.522
C07234=1184.334,332.529,-74.059,-176.400,8.061,148.522
C07235=1184.338,332.282,-74.025,-176.402,8.057,148.522
C07236=1184.342,332.034,-73.994,-176.405,8.054,148.522
C07237=1184.346,331.786,-73.962,-176.407,8.051,148.521
C07238=1184.351,331.538,-73.930,-176.410,8.048,148.521
C07239=1184.355,331.290,-73.898,-176.412,8.045,148.521
C07240=1184.360,331.042,-73.866,-176.415,8.041,148.521
C07241=1184.363,330.794,-73.834,-176.417,8.038,148.521
C07242=1184.367,330.546,-73.802,-176.420,8.035,148.521
C07243=1184.371,330.298,-73.770,-176.422,8.032,148.521
C07244=1184.376,330.050,-73.738,-176.424,8.029,148.521
C07245=1184.380,329.802,-73.706,-176.427,8.025,148.520
C07246=1184.384,329.554,-73.674,-176.428,8.023,148.520
C07247=1184.388,329.307,-73.642,-176.431,8.020,148.520
C07248=1184.393,329.058,-73.610,-176.433,8.017,148.520
C07249=1184.396,328.810,-73.578,-176.436,8.014,148.520
C07250=1184.401,328.563,-73.547,-176.438,8.010,148.520
C07251=1184.405,328.315,-73.514,-176.441,8.007,148.520
C07252=1184.409,328.067,-73.482,-176.443,8.004,148.520
C07253=1184.413,327.819,-73.451,-176.446,8.001,148.519
C07254=1184.417,327.571,-73.419,-176.448,7.998,148.519
C07255=1184.422,327.324,-73.387,-176.451,7.994,148.519
C07256=1184.426,327.076,-73.355,-176.453,7.991,148.519
C07257=1184.429,326.828,-73.323,-176.456,7.988,148.519
C07258=1184.434,326.580,-73.291,-176.458,7.985,148.519
C07259=1184.438,326.331,-73.260,-176.460,7.982,148.519
C07260=1184.442,326.083,-73.228,-176.463,7.980,148.519
C07261=1184.446,325.836,-73.197,-176.465,7.976,148.519
C07262=1184.450,325.588,-73.165,-176.468,7.973,148.519
C07263=1184.455,325.340,-73.133,-176.470,7.970,148.518
C07264=1184.459,325.091,-73.102,-176.472,7.967,148.518
C07265=1184.463,324.843,-73.070,-176.475,7.964,148.518
C07266=1184.467,324.596,-73.038,-176.477,7.960,148.518
C07267=1184.471,324.348,-73.006,-176.480,7.957,148.518
C07268=1184.476,324.100,-72.975,-176.483,7.954,148.518
C07269=1184.480,323.852,-72.943,-176.485,7.951,148.518
C07270=1184.484,323.604,-72.912,-176.487,7.948,148.518
C07271=1184.488,323.356,-72.881,-176.490,7.945,148.518
C07272=1184.492,323.108,-72.849,-176.492,7.942,148.518
C07273=1184.496,322.860,-72.817,-176.494,7.939,148.518
C07274=1184.500,322.612,-72.786,-176.497,7.936,148.518
C07275=1184.505,322.364,-72.755,-176.499,7.933,148.517
C07276=1184.509,322.116,-72.722,-176.502,7.930,148.517
C07277=1184.514,321.868,-72.692,-176.504,7.926,148.517
C07278=1184.517,321.620,-72.660,-176.507,7.923,148.517
C07279=1184.522,321.372,-72.629,-176.509,7.920,148.517
C07280=1184.526,321.124,-72.597,-176.512,7.917,148.517
C07281=1184.530,320.877,-72.566,-176.514,7.914,148.517
C07282=1184.534,320.628,-72.534,-176.516,7.912,148.517
C07283=1184.538,320.381,-72.503,-176.519,7.909,148.517
C07284=1184.542,320.132,-72.472,-176.521,7.905,148.517
C07285=1184.547,319.885,-72.440,-176.524,7.902,148.517
C07286=1184.551,319.636,-72.409,-176.526,7.899,148.516
C07287=1184.555,319.389,-72.378,-176.529,7.896,148.516
C07288=1184.559,319.140,-72.347,-176.532,7.893,148.516
C07289=1184.563,318.893,-72.315,-176.534,7.890,148.516
C07290=1184.567,318.644,-72.284,-176.536,7.887,148.516
C07291=1184.572,318.396,-72.253,-176.539,7.883,148.516
C07292=1184.576,318.148,-72.221,-176.541,7.881,148.516
C07293=1184.580,317.900,-72.191,-176.544,7.878,148.516
C07294=1184.585,317.653,-72.159,-176.546,7.875,148.516
C07295=1184.589,317.404,-72.128,-176.549,7.872,148.516
C07296=1184.593,317.156,-72.097,-176.551,7.869,148.516
C07297=1184.597,316.908,-72.065,-176.554,7.866,148.516
C07298=1184.601,316.660,-72.035,-176.556,7.863,148.516
C07299=1184.605,316.411,-72.004,-176.558,7.859,148.515
C07300=1184.609,316.164,-71.973,-176.561,7.856,148.516
C07301=1184.614,315.917,-71.942,-176.563,7.854,148.516
C07302=1184.618,315.668,-71.911,-176.566,7.851,148.515
C07303=1184.622,315.420,-71.880,-176.568,7.848,148.515
C07304=1184.626,315.172,-71.848,-176.571,7.845,148.515
C07305=1184.631,314.924,-71.817,-176.573,7.841,148.515
C07306=1184.635,314.647,-71.783,-176.576,7.838,148.515
C07307=1184.641,314.371,-71.749,-176.579,7.835,148.515
C07308=1184.645,314.094,-71.714,-176.582,7.831,148.515
C07309=1184.649,313.818,-71.679,-176.584,7.828,148.515
C07310=1184.654,313.570,-71.649,-176.587,7.825,148.515
C07311=1184.658,313.321,-71.617,-176.590,7.822,148.515
